Fanuc TP program (LS listing): 190220_hosenrohr_oV2.ls

/PROG  190220_hosenrohr_oV2
/ATTR
COMMENT	= "19-02-22 10:03:29";
PROG_SIZE	= 0;
DEFAULT_GROUP	= 1, 1, *, *, *;
/APPL
    ARC Welding Equipment: 1, *, *, *, *;
/MN
   1:  CALL HOME_ALL;
   1:  UFRAME_NUM = 1;
   1:  UTOOL_NUM = 3;
   1:  COL GUARD ADJUST 150;
   1:  ! -- Layer/Ebene 62 -- !;
   1:  PR[91] = PR[90];
   1:  PR[GP1:91,1] = PR[GP1:90,1] + -0.384;
   1:  PR[GP1:91,2] = PR[GP1:90,2] + 18.027;
   1:  PR[GP1:91,3] = PR[GP1:90,3] + 38.125;
   1:  !Sicherheitspunkt!;
   1:  PR[92] = PR[91];
   1:  PR[92] = PR[GP1:92,3] + 50;
   1:J PR[92];
   1:  !Schweissanfang anfahren!;
   1:L PR[91] R[100]mm/sec CNT100;
   1:  CALL LASER_DRAHT_START;
   1:  PR[GP1:91,1] = PR[GP1:90,1] + -4.016;
   1:  PR[GP1:91,2] = PR[GP1:90,2] + 19.874;
   1:L PR[91] R[100]mm/sec CNT100;
   1:  PR[GP1:91,1] = PR[GP1:90,1] + -8.099;
   1:  PR[GP1:91,2] = PR[GP1:90,2] + 24.627;
   1:L PR[91] R[100]mm/sec CNT100;
   1:  PR[GP1:91,1] = PR[GP1:90,1] + -13.957;
   1:  PR[GP1:91,2] = PR[GP1:90,2] + 29.191;
   1:L PR[91] R[100]mm/sec CNT100;
   1:  PR[GP1:91,1] = PR[GP1:90,1] + -18.277;
   1:  PR[GP1:91,2] = PR[GP1:90,2] + 31.547;
   1:L PR[91] R[100]mm/sec CNT100;
   1:  PR[GP1:91,1] = PR[GP1:90,1] + -22.719;
   1:  PR[GP1:91,2] = PR[GP1:90,2] + 33.113;
   1:L PR[91] R[100]mm/sec CNT100;
   1:  PR[GP1:91,1] = PR[GP1:90,1] + -26.359;
   1:  PR[GP1:91,2] = PR[GP1:90,2] + 34.297;
   1:L PR[91] R[100]mm/sec CNT100;
   1:  PR[GP1:91,1] = PR[GP1:90,1] + -28.832;
   1:  PR[GP1:91,2] = PR[GP1:90,2] + 34.657;
   1:L PR[91] R[100]mm/sec CNT100;
   1:  PR[GP1:91,1] = PR[GP1:90,1] + -36.965;
   1:  PR[GP1:91,2] = PR[GP1:90,2] + 35.069;
   1:L PR[91] R[100]mm/sec CNT100;
   1:  PR[GP1:91,1] = PR[GP1:90,1] + -38.092;
   1:  PR[GP1:91,2] = PR[GP1:90,2] + 35.037;
   1:L PR[91] R[100]mm/sec CNT100;
   1:  PR[GP1:91,1] = PR[GP1:90,1] + -45.127;
   1:  PR[GP1:91,2] = PR[GP1:90,2] + 33.402;
   1:L PR[91] R[100]mm/sec CNT100;
   1:  PR[GP1:91,1] = PR[GP1:90,1] + -48.487;
   1:  PR[GP1:91,2] = PR[GP1:90,2] + 32.649;
   1:L PR[91] R[100]mm/sec CNT100;
   1:  PR[GP1:91,1] = PR[GP1:90,1] + -49.175;
   1:  PR[GP1:91,2] = PR[GP1:90,2] + 32.303;
   1:L PR[91] R[100]mm/sec CNT100;
   1:  PR[GP1:91,1] = PR[GP1:90,1] + -57.619;
   1:  PR[GP1:91,2] = PR[GP1:90,2] + 27.543;
   1:L PR[91] R[100]mm/sec CNT100;
   1:  PR[GP1:91,1] = PR[GP1:90,1] + -59.619;
   1:  PR[GP1:91,2] = PR[GP1:90,2] + 25.581;
   1:L PR[91] R[100]mm/sec CNT100;
   1:  PR[GP1:91,1] = PR[GP1:90,1] + -64.977;
   1:  PR[GP1:91,2] = PR[GP1:90,2] + 19.937;
   1:L PR[91] R[100]mm/sec CNT100;
   1:  PR[GP1:91,1] = PR[GP1:90,1] + -66.878;
   1:  PR[GP1:91,2] = PR[GP1:90,2] + 16.287;
   1:L PR[91] R[100]mm/sec CNT100;
   1:  PR[GP1:91,1] = PR[GP1:90,1] + -69.759;
   1:  PR[GP1:91,2] = PR[GP1:90,2] + 10.455;
   1:L PR[91] R[100]mm/sec CNT100;
   1:  PR[GP1:91,1] = PR[GP1:90,1] + -70.528;
   1:  PR[GP1:91,2] = PR[GP1:90,2] + 5.716;
   1:L PR[91] R[100]mm/sec CNT100;
   1:  PR[GP1:91,1] = PR[GP1:90,1] + -70.620;
   1:  PR[GP1:91,2] = PR[GP1:90,2] + 5.247;
   1:L PR[91] R[100]mm/sec CNT100;
   1:  PR[GP1:91,1] = PR[GP1:90,1] + -71.434;
   1:  PR[GP1:91,2] = PR[GP1:90,2] + -0.068;
   1:L PR[91] R[100]mm/sec CNT100;
   1:  PR[GP1:91,1] = PR[GP1:90,1] + -70.618;
   1:  PR[GP1:91,2] = PR[GP1:90,2] + -4.964;
   1:L PR[91] R[100]mm/sec CNT100;
   1:  PR[GP1:91,1] = PR[GP1:90,1] + -69.758;
   1:  PR[GP1:91,2] = PR[GP1:90,2] + -10.601;
   1:L PR[91] R[100]mm/sec CNT100;
   1:  PR[GP1:91,1] = PR[GP1:90,1] + -66.878;
   1:  PR[GP1:91,2] = PR[GP1:90,2] + -16.431;
   1:L PR[91] R[100]mm/sec CNT100;
   1:  PR[GP1:91,1] = PR[GP1:90,1] + -64.977;
   1:  PR[GP1:91,2] = PR[GP1:90,2] + -20.081;
   1:L PR[91] R[100]mm/sec CNT100;
   1:  PR[GP1:91,1] = PR[GP1:90,1] + -59.619;
   1:  PR[GP1:91,2] = PR[GP1:90,2] + -25.725;
   1:L PR[91] R[100]mm/sec CNT100;
   1:  PR[GP1:91,1] = PR[GP1:90,1] + -57.619;
   1:  PR[GP1:91,2] = PR[GP1:90,2] + -27.687;
   1:L PR[91] R[100]mm/sec CNT100;
   1:  PR[GP1:91,1] = PR[GP1:90,1] + -49.175;
   1:  PR[GP1:91,2] = PR[GP1:90,2] + -32.447;
   1:L PR[91] R[100]mm/sec CNT100;
   1:  PR[GP1:91,1] = PR[GP1:90,1] + -48.487;
   1:  PR[GP1:91,2] = PR[GP1:90,2] + -32.793;
   1:L PR[91] R[100]mm/sec CNT100;
   1:  PR[GP1:91,1] = PR[GP1:90,1] + -45.126;
   1:  PR[GP1:91,2] = PR[GP1:90,2] + -33.546;
   1:L PR[91] R[100]mm/sec CNT100;
   1:  PR[GP1:91,1] = PR[GP1:90,1] + -38.859;
   1:  PR[GP1:91,2] = PR[GP1:90,2] + -35.021;
   1:L PR[91] R[100]mm/sec CNT100;
   1:  PR[GP1:91,1] = PR[GP1:90,1] + -38.098;
   1:  PR[GP1:91,2] = PR[GP1:90,2] + -35.181;
   1:L PR[91] R[100]mm/sec CNT100;
   1:  PR[GP1:91,1] = PR[GP1:90,1] + -36.965;
   1:  PR[GP1:91,2] = PR[GP1:90,2] + -35.213;
   1:L PR[91] R[100]mm/sec CNT100;
   1:  PR[GP1:91,1] = PR[GP1:90,1] + -28.832;
   1:  PR[GP1:91,2] = PR[GP1:90,2] + -34.801;
   1:L PR[91] R[100]mm/sec CNT100;
   1:  PR[GP1:91,1] = PR[GP1:90,1] + -26.368;
   1:  PR[GP1:91,2] = PR[GP1:90,2] + -34.443;
   1:L PR[91] R[100]mm/sec CNT100;
   1:  PR[GP1:91,1] = PR[GP1:90,1] + -21.518;
   1:  PR[GP1:91,2] = PR[GP1:90,2] + -32.707;
   1:L PR[91] R[100]mm/sec CNT100;
   1:  PR[GP1:91,1] = PR[GP1:90,1] + -18.268;
   1:  PR[GP1:91,2] = PR[GP1:90,2] + -31.686;
   1:L PR[91] R[100]mm/sec CNT100;
   1:  PR[GP1:91,1] = PR[GP1:90,1] + -13.949;
   1:  PR[GP1:91,2] = PR[GP1:90,2] + -29.331;
   1:L PR[91] R[100]mm/sec CNT100;
   1:  PR[GP1:91,1] = PR[GP1:90,1] + -12.372;
   1:  PR[GP1:91,2] = PR[GP1:90,2] + -28.176;
   1:L PR[91] R[100]mm/sec CNT100;
   1:  PR[GP1:91,1] = PR[GP1:90,1] + -8.101;
   1:  PR[GP1:91,2] = PR[GP1:90,2] + -24.773;
   1:L PR[91] R[100]mm/sec CNT100;
   1:  PR[GP1:91,1] = PR[GP1:90,1] + -3.961;
   1:  PR[GP1:91,2] = PR[GP1:90,2] + -19.964;
   1:L PR[91] R[100]mm/sec CNT100;
   1:  PR[GP1:91,1] = PR[GP1:90,1] + -3.637;
   1:  PR[GP1:91,2] = PR[GP1:90,2] + -19.895;
   1:L PR[91] R[100]mm/sec CNT100;
   1:  PR[GP1:91,1] = PR[GP1:90,1] + 0.136;
   1:  PR[GP1:91,2] = PR[GP1:90,2] + -17.894;
   1:L PR[91] R[100]mm/sec CNT100;
   1:  PR[GP1:91,1] = PR[GP1:90,1] + 0.611;
   1:  PR[GP1:91,2] = PR[GP1:90,2] + -18.171;
   1:L PR[91] R[100]mm/sec CNT100;
   1:  PR[GP1:91,1] = PR[GP1:90,1] + 4.242;
   1:  PR[GP1:91,2] = PR[GP1:90,2] + -20.026;
   1:L PR[91] R[100]mm/sec CNT100;
   1:  PR[GP1:91,1] = PR[GP1:90,1] + 8.362;
   1:  PR[GP1:91,2] = PR[GP1:90,2] + -24.817;
   1:L PR[91] R[100]mm/sec CNT100;
   1:  PR[GP1:91,1] = PR[GP1:90,1] + 14.189;
   1:  PR[GP1:91,2] = PR[GP1:90,2] + -29.353;
   1:L PR[91] R[100]mm/sec CNT100;
   1:  PR[GP1:91,1] = PR[GP1:90,1] + 18.481;
   1:  PR[GP1:91,2] = PR[GP1:90,2] + -31.687;
   1:L PR[91] R[100]mm/sec CNT100;
   1:  PR[GP1:91,1] = PR[GP1:90,1] + 22.922;
   1:  PR[GP1:91,2] = PR[GP1:90,2] + -33.252;
   1:L PR[91] R[100]mm/sec CNT100;
   1:  PR[GP1:91,1] = PR[GP1:90,1] + 26.570;
   1:  PR[GP1:91,2] = PR[GP1:90,2] + -34.439;
   1:L PR[91] R[100]mm/sec CNT100;
   1:  PR[GP1:91,1] = PR[GP1:90,1] + 29.041;
   1:  PR[GP1:91,2] = PR[GP1:90,2] + -34.800;
   1:L PR[91] R[100]mm/sec CNT100;
   1:  PR[GP1:91,1] = PR[GP1:90,1] + 37.175;
   1:  PR[GP1:91,2] = PR[GP1:90,2] + -35.214;
   1:L PR[91] R[100]mm/sec CNT100;
   1:  PR[GP1:91,1] = PR[GP1:90,1] + 38.299;
   1:  PR[GP1:91,2] = PR[GP1:90,2] + -35.183;
   1:L PR[91] R[100]mm/sec CNT100;
   1:  PR[GP1:91,1] = PR[GP1:90,1] + 45.340;
   1:  PR[GP1:91,2] = PR[GP1:90,2] + -33.544;
   1:L PR[91] R[100]mm/sec CNT100;
   1:  PR[GP1:91,1] = PR[GP1:90,1] + 48.700;
   1:  PR[GP1:91,2] = PR[GP1:90,2] + -32.790;
   1:L PR[91] R[100]mm/sec CNT100;
   1:  PR[GP1:91,1] = PR[GP1:90,1] + 49.388;
   1:  PR[GP1:91,2] = PR[GP1:90,2] + -32.445;
   1:L PR[91] R[100]mm/sec CNT100;
   1:  PR[GP1:91,1] = PR[GP1:90,1] + 57.830;
   1:  PR[GP1:91,2] = PR[GP1:90,2] + -27.694;
   1:L PR[91] R[100]mm/sec CNT100;
   1:  PR[GP1:91,1] = PR[GP1:90,1] + 59.830;
   1:  PR[GP1:91,2] = PR[GP1:90,2] + -25.729;
   1:L PR[91] R[100]mm/sec CNT100;
   1:  PR[GP1:91,1] = PR[GP1:90,1] + 65.189;
   1:  PR[GP1:91,2] = PR[GP1:90,2] + -20.068;
   1:L PR[91] R[100]mm/sec CNT100;
   1:  PR[GP1:91,1] = PR[GP1:90,1] + 67.091;
   1:  PR[GP1:91,2] = PR[GP1:90,2] + -16.427;
   1:L PR[91] R[100]mm/sec CNT100;
   1:  PR[GP1:91,1] = PR[GP1:90,1] + 69.972;
   1:  PR[GP1:91,2] = PR[GP1:90,2] + -10.623;
   1:L PR[91] R[100]mm/sec CNT100;
   1:  PR[GP1:91,1] = PR[GP1:90,1] + 70.741;
   1:  PR[GP1:91,2] = PR[GP1:90,2] + -5.877;
   1:L PR[91] R[100]mm/sec CNT100;
   1:  PR[GP1:91,1] = PR[GP1:90,1] + 70.833;
   1:  PR[GP1:91,2] = PR[GP1:90,2] + -5.406;
   1:L PR[91] R[100]mm/sec CNT100;
   1:  PR[GP1:91,1] = PR[GP1:90,1] + 71.648;
   1:  PR[GP1:91,2] = PR[GP1:90,2] + -0.076;
   1:L PR[91] R[100]mm/sec CNT100;
   1:  PR[GP1:91,1] = PR[GP1:90,1] + 70.831;
   1:  PR[GP1:91,2] = PR[GP1:90,2] + 4.828;
   1:L PR[91] R[100]mm/sec CNT100;
   1:  PR[GP1:91,1] = PR[GP1:90,1] + 69.971;
   1:  PR[GP1:91,2] = PR[GP1:90,2] + 10.481;
   1:L PR[91] R[100]mm/sec CNT100;
   1:  PR[GP1:91,1] = PR[GP1:90,1] + 67.091;
   1:  PR[GP1:91,2] = PR[GP1:90,2] + 16.283;
   1:L PR[91] R[100]mm/sec CNT100;
   1:  PR[GP1:91,1] = PR[GP1:90,1] + 65.189;
   1:  PR[GP1:91,2] = PR[GP1:90,2] + 19.924;
   1:L PR[91] R[100]mm/sec CNT100;
   1:  PR[GP1:91,1] = PR[GP1:90,1] + 59.830;
   1:  PR[GP1:91,2] = PR[GP1:90,2] + 25.585;
   1:L PR[91] R[100]mm/sec CNT100;
   1:  PR[GP1:91,1] = PR[GP1:90,1] + 57.830;
   1:  PR[GP1:91,2] = PR[GP1:90,2] + 27.550;
   1:L PR[91] R[100]mm/sec CNT100;
   1:  PR[GP1:91,1] = PR[GP1:90,1] + 49.388;
   1:  PR[GP1:91,2] = PR[GP1:90,2] + 32.301;
   1:L PR[91] R[100]mm/sec CNT100;
   1:  PR[GP1:91,1] = PR[GP1:90,1] + 48.700;
   1:  PR[GP1:91,2] = PR[GP1:90,2] + 32.646;
   1:L PR[91] R[100]mm/sec CNT100;
   1:  PR[GP1:91,1] = PR[GP1:90,1] + 45.339;
   1:  PR[GP1:91,2] = PR[GP1:90,2] + 33.400;
   1:L PR[91] R[100]mm/sec CNT100;
   1:  PR[GP1:91,1] = PR[GP1:90,1] + 39.068;
   1:  PR[GP1:91,2] = PR[GP1:90,2] + 34.879;
   1:L PR[91] R[100]mm/sec CNT100;
   1:  PR[GP1:91,1] = PR[GP1:90,1] + 38.306;
   1:  PR[GP1:91,2] = PR[GP1:90,2] + 35.039;
   1:L PR[91] R[100]mm/sec CNT100;
   1:  PR[GP1:91,1] = PR[GP1:90,1] + 37.175;
   1:  PR[GP1:91,2] = PR[GP1:90,2] + 35.070;
   1:L PR[91] R[100]mm/sec CNT100;
   1:  PR[GP1:91,1] = PR[GP1:90,1] + 29.041;
   1:  PR[GP1:91,2] = PR[GP1:90,2] + 34.656;
   1:L PR[91] R[100]mm/sec CNT100;
   1:  PR[GP1:91,1] = PR[GP1:90,1] + 26.579;
   1:  PR[GP1:91,2] = PR[GP1:90,2] + 34.296;
   1:L PR[91] R[100]mm/sec CNT100;
   1:  PR[GP1:91,1] = PR[GP1:90,1] + 21.729;
   1:  PR[GP1:91,2] = PR[GP1:90,2] + 32.563;
   1:L PR[91] R[100]mm/sec CNT100;
   1:  PR[GP1:91,1] = PR[GP1:90,1] + 18.472;
   1:  PR[GP1:91,2] = PR[GP1:90,2] + 31.539;
   1:L PR[91] R[100]mm/sec CNT100;
   1:  PR[GP1:91,1] = PR[GP1:90,1] + 14.182;
   1:  PR[GP1:91,2] = PR[GP1:90,2] + 29.205;
   1:L PR[91] R[100]mm/sec CNT100;
   1:  PR[GP1:91,1] = PR[GP1:90,1] + 12.601;
   1:  PR[GP1:91,2] = PR[GP1:90,2] + 28.047;
   1:L PR[91] R[100]mm/sec CNT100;
   1:  PR[GP1:91,1] = PR[GP1:90,1] + 8.365;
   1:  PR[GP1:91,2] = PR[GP1:90,2] + 24.676;
   1:L PR[91] R[100]mm/sec CNT100;
   1:  PR[GP1:91,1] = PR[GP1:90,1] + 4.242;
   1:  PR[GP1:91,2] = PR[GP1:90,2] + 19.873;
   1:L PR[91] R[100]mm/sec CNT100;
   1:  PR[GP1:91,1] = PR[GP1:90,1] + 0.084;
   1:  PR[GP1:91,2] = PR[GP1:90,2] + 17.753;
   1:L PR[91] R[100]mm/sec CNT100;
   1:  ! -- Layer/Ebene 63 -- !;
   1:  PR[91] = PR[90];
   1:  PR[GP1:91,1] = PR[GP1:90,1] + -0.147;
   1:  PR[GP1:91,2] = PR[GP1:90,2] + 18.208;
   1:  PR[GP1:91,3] = PR[GP1:90,3] + 38.735;
   1:L PR[91] R[100]mm/sec CNT100;
   1:  PR[GP1:91,1] = PR[GP1:90,1] + -3.986;
   1:  PR[GP1:91,2] = PR[GP1:90,2] + 20.161;
   1:L PR[91] R[100]mm/sec CNT100;
   1:  PR[GP1:91,1] = PR[GP1:90,1] + -7.934;
   1:  PR[GP1:91,2] = PR[GP1:90,2] + 24.750;
   1:L PR[91] R[100]mm/sec CNT100;
   1:  PR[GP1:91,1] = PR[GP1:90,1] + -13.454;
   1:  PR[GP1:91,2] = PR[GP1:90,2] + 29.065;
   1:L PR[91] R[100]mm/sec CNT100;
   1:  PR[GP1:91,1] = PR[GP1:90,1] + -18.260;
   1:  PR[GP1:91,2] = PR[GP1:90,2] + 31.685;
   1:L PR[91] R[100]mm/sec CNT100;
   1:  PR[GP1:91,1] = PR[GP1:90,1] + -21.778;
   1:  PR[GP1:91,2] = PR[GP1:90,2] + 32.926;
   1:L PR[91] R[100]mm/sec CNT100;
   1:  PR[GP1:91,1] = PR[GP1:90,1] + -26.058;
   1:  PR[GP1:91,2] = PR[GP1:90,2] + 34.319;
   1:L PR[91] R[100]mm/sec CNT100;
   1:  PR[GP1:91,1] = PR[GP1:90,1] + -28.972;
   1:  PR[GP1:91,2] = PR[GP1:90,2] + 34.743;
   1:L PR[91] R[100]mm/sec CNT100;
   1:  PR[GP1:91,1] = PR[GP1:90,1] + -36.314;
   1:  PR[GP1:91,2] = PR[GP1:90,2] + 35.115;
   1:L PR[91] R[100]mm/sec CNT100;
   1:  PR[GP1:91,1] = PR[GP1:90,1] + -37.972;
   1:  PR[GP1:91,2] = PR[GP1:90,2] + 35.068;
   1:L PR[91] R[100]mm/sec CNT100;
   1:  PR[GP1:91,1] = PR[GP1:90,1] + -48.463;
   1:  PR[GP1:91,2] = PR[GP1:90,2] + 32.632;
   1:L PR[91] R[100]mm/sec CNT100;
   1:  PR[GP1:91,1] = PR[GP1:90,1] + -57.569;
   1:  PR[GP1:91,2] = PR[GP1:90,2] + 27.505;
   1:L PR[91] R[100]mm/sec CNT100;
   1:  PR[GP1:91,1] = PR[GP1:90,1] + -59.075;
   1:  PR[GP1:91,2] = PR[GP1:90,2] + 26.027;
   1:L PR[91] R[100]mm/sec CNT100;
   1:  PR[GP1:91,1] = PR[GP1:90,1] + -64.892;
   1:  PR[GP1:91,2] = PR[GP1:90,2] + 19.900;
   1:L PR[91] R[100]mm/sec CNT100;
   1:  PR[GP1:91,1] = PR[GP1:90,1] + -66.497;
   1:  PR[GP1:91,2] = PR[GP1:90,2] + 16.818;
   1:L PR[91] R[100]mm/sec CNT100;
   1:  PR[GP1:91,1] = PR[GP1:90,1] + -69.651;
   1:  PR[GP1:91,2] = PR[GP1:90,2] + 10.434;
   1:L PR[91] R[100]mm/sec CNT100;
   1:  PR[GP1:91,1] = PR[GP1:90,1] + -70.323;
   1:  PR[GP1:91,2] = PR[GP1:90,2] + 6.290;
   1:L PR[91] R[100]mm/sec CNT100;
   1:  PR[GP1:91,1] = PR[GP1:90,1] + -70.403;
   1:  PR[GP1:91,2] = PR[GP1:90,2] + 5.879;
   1:L PR[91] R[100]mm/sec CNT100;
   1:  PR[GP1:91,1] = PR[GP1:90,1] + -71.315;
   1:  PR[GP1:91,2] = PR[GP1:90,2] + -0.068;
   1:L PR[91] R[100]mm/sec CNT100;
   1:  PR[GP1:91,1] = PR[GP1:90,1] + -70.592;
   1:  PR[GP1:91,2] = PR[GP1:90,2] + -4.409;
   1:L PR[91] R[100]mm/sec CNT100;
   1:  PR[GP1:91,1] = PR[GP1:90,1] + -69.650;
   1:  PR[GP1:91,2] = PR[GP1:90,2] + -10.580;
   1:L PR[91] R[100]mm/sec CNT100;
   1:  PR[GP1:91,1] = PR[GP1:90,1] + -66.497;
   1:  PR[GP1:91,2] = PR[GP1:90,2] + -16.962;
   1:L PR[91] R[100]mm/sec CNT100;
   1:  PR[GP1:91,1] = PR[GP1:90,1] + -64.892;
   1:  PR[GP1:91,2] = PR[GP1:90,2] + -20.044;
   1:L PR[91] R[100]mm/sec CNT100;
   1:  PR[GP1:91,1] = PR[GP1:90,1] + -59.075;
   1:  PR[GP1:91,2] = PR[GP1:90,2] + -26.171;
   1:L PR[91] R[100]mm/sec CNT100;
   1:  PR[GP1:91,1] = PR[GP1:90,1] + -57.569;
   1:  PR[GP1:91,2] = PR[GP1:90,2] + -27.649;
   1:L PR[91] R[100]mm/sec CNT100;
   1:  PR[GP1:91,1] = PR[GP1:90,1] + -48.463;
   1:  PR[GP1:91,2] = PR[GP1:90,2] + -32.777;
   1:L PR[91] R[100]mm/sec CNT100;
   1:  PR[GP1:91,1] = PR[GP1:90,1] + -39.099;
   1:  PR[GP1:91,2] = PR[GP1:90,2] + -34.975;
   1:L PR[91] R[100]mm/sec CNT100;
   1:  PR[GP1:91,1] = PR[GP1:90,1] + -37.979;
   1:  PR[GP1:91,2] = PR[GP1:90,2] + -35.211;
   1:L PR[91] R[100]mm/sec CNT100;
   1:  PR[GP1:91,1] = PR[GP1:90,1] + -36.314;
   1:  PR[GP1:91,2] = PR[GP1:90,2] + -35.259;
   1:L PR[91] R[100]mm/sec CNT100;
   1:  PR[GP1:91,1] = PR[GP1:90,1] + -28.972;
   1:  PR[GP1:91,2] = PR[GP1:90,2] + -34.887;
   1:L PR[91] R[100]mm/sec CNT100;
   1:  PR[GP1:91,1] = PR[GP1:90,1] + -26.066;
   1:  PR[GP1:91,2] = PR[GP1:90,2] + -34.464;
   1:L PR[91] R[100]mm/sec CNT100;
   1:  PR[GP1:91,1] = PR[GP1:90,1] + -21.865;
   1:  PR[GP1:91,2] = PR[GP1:90,2] + -32.960;
   1:L PR[91] R[100]mm/sec CNT100;
   1:  PR[GP1:91,1] = PR[GP1:90,1] + -18.251;
   1:  PR[GP1:91,2] = PR[GP1:90,2] + -31.824;
   1:L PR[91] R[100]mm/sec CNT100;
   1:  PR[GP1:91,1] = PR[GP1:90,1] + -13.445;
   1:  PR[GP1:91,2] = PR[GP1:90,2] + -29.204;
   1:L PR[91] R[100]mm/sec CNT100;
   1:  PR[GP1:91,1] = PR[GP1:90,1] + -12.545;
   1:  PR[GP1:91,2] = PR[GP1:90,2] + -28.544;
   1:L PR[91] R[100]mm/sec CNT100;
   1:  PR[GP1:91,1] = PR[GP1:90,1] + -9.672;
   1:  PR[GP1:91,2] = PR[GP1:90,2] + -26.256;
   1:L PR[91] R[100]mm/sec CNT100;
   1:  PR[GP1:91,1] = PR[GP1:90,1] + -7.920;
   1:  PR[GP1:91,2] = PR[GP1:90,2] + -24.884;
   1:L PR[91] R[100]mm/sec CNT100;
   1:  PR[GP1:91,1] = PR[GP1:90,1] + -3.931;
   1:  PR[GP1:91,2] = PR[GP1:90,2] + -20.257;
   1:L PR[91] R[100]mm/sec CNT100;
   1:  PR[GP1:91,1] = PR[GP1:90,1] + -3.470;
   1:  PR[GP1:91,2] = PR[GP1:90,2] + -20.158;
   1:L PR[91] R[100]mm/sec CNT100;
   1:  PR[GP1:91,1] = PR[GP1:90,1] + 0.146;
   1:  PR[GP1:91,2] = PR[GP1:90,2] + -18.242;
   1:L PR[91] R[100]mm/sec CNT100;
   1:  PR[GP1:91,1] = PR[GP1:90,1] + 4.212;
   1:  PR[GP1:91,2] = PR[GP1:90,2] + -20.319;
   1:L PR[91] R[100]mm/sec CNT100;
   1:  PR[GP1:91,1] = PR[GP1:90,1] + 8.183;
   1:  PR[GP1:91,2] = PR[GP1:90,2] + -24.930;
   1:L PR[91] R[100]mm/sec CNT100;
   1:  PR[GP1:91,1] = PR[GP1:90,1] + 13.688;
   1:  PR[GP1:91,2] = PR[GP1:90,2] + -29.229;
   1:L PR[91] R[100]mm/sec CNT100;
   1:  PR[GP1:91,1] = PR[GP1:90,1] + 18.463;
   1:  PR[GP1:91,2] = PR[GP1:90,2] + -31.826;
   1:L PR[91] R[100]mm/sec CNT100;
   1:  PR[GP1:91,1] = PR[GP1:90,1] + 21.979;
   1:  PR[GP1:91,2] = PR[GP1:90,2] + -33.064;
   1:L PR[91] R[100]mm/sec CNT100;
   1:  PR[GP1:91,1] = PR[GP1:90,1] + 26.268;
   1:  PR[GP1:91,2] = PR[GP1:90,2] + -34.460;
   1:L PR[91] R[100]mm/sec CNT100;
   1:  PR[GP1:91,1] = PR[GP1:90,1] + 29.180;
   1:  PR[GP1:91,2] = PR[GP1:90,2] + -34.886;
   1:L PR[91] R[100]mm/sec CNT100;
   1:  PR[GP1:91,1] = PR[GP1:90,1] + 36.523;
   1:  PR[GP1:91,2] = PR[GP1:90,2] + -35.259;
   1:L PR[91] R[100]mm/sec CNT100;
   1:  PR[GP1:91,1] = PR[GP1:90,1] + 38.177;
   1:  PR[GP1:91,2] = PR[GP1:90,2] + -35.213;
   1:L PR[91] R[100]mm/sec CNT100;
   1:  PR[GP1:91,1] = PR[GP1:90,1] + 48.676;
   1:  PR[GP1:91,2] = PR[GP1:90,2] + -32.773;
   1:L PR[91] R[100]mm/sec CNT100;
   1:  PR[GP1:91,1] = PR[GP1:90,1] + 57.781;
   1:  PR[GP1:91,2] = PR[GP1:90,2] + -27.655;
   1:L PR[91] R[100]mm/sec CNT100;
   1:  PR[GP1:91,1] = PR[GP1:90,1] + 59.287;
   1:  PR[GP1:91,2] = PR[GP1:90,2] + -26.175;
   1:L PR[91] R[100]mm/sec CNT100;
   1:  PR[GP1:91,1] = PR[GP1:90,1] + 65.104;
   1:  PR[GP1:91,2] = PR[GP1:90,2] + -20.031;
   1:L PR[91] R[100]mm/sec CNT100;
   1:  PR[GP1:91,1] = PR[GP1:90,1] + 66.710;
   1:  PR[GP1:91,2] = PR[GP1:90,2] + -16.955;
   1:L PR[91] R[100]mm/sec CNT100;
   1:  PR[GP1:91,1] = PR[GP1:90,1] + 69.864;
   1:  PR[GP1:91,2] = PR[GP1:90,2] + -10.602;
   1:L PR[91] R[100]mm/sec CNT100;
   1:  PR[GP1:91,1] = PR[GP1:90,1] + 70.536;
   1:  PR[GP1:91,2] = PR[GP1:90,2] + -6.453;
   1:L PR[91] R[100]mm/sec CNT100;
   1:  PR[GP1:91,1] = PR[GP1:90,1] + 70.616;
   1:  PR[GP1:91,2] = PR[GP1:90,2] + -6.041;
   1:L PR[91] R[100]mm/sec CNT100;
   1:  PR[GP1:91,1] = PR[GP1:90,1] + 71.528;
   1:  PR[GP1:91,2] = PR[GP1:90,2] + -0.076;
   1:L PR[91] R[100]mm/sec CNT100;
   1:  PR[GP1:91,1] = PR[GP1:90,1] + 70.804;
   1:  PR[GP1:91,2] = PR[GP1:90,2] + 4.273;
   1:L PR[91] R[100]mm/sec CNT100;
   1:  PR[GP1:91,1] = PR[GP1:90,1] + 69.862;
   1:  PR[GP1:91,2] = PR[GP1:90,2] + 10.461;
   1:L PR[91] R[100]mm/sec CNT100;
   1:  PR[GP1:91,1] = PR[GP1:90,1] + 66.710;
   1:  PR[GP1:91,2] = PR[GP1:90,2] + 16.811;
   1:L PR[91] R[100]mm/sec CNT100;
   1:  PR[GP1:91,1] = PR[GP1:90,1] + 65.104;
   1:  PR[GP1:91,2] = PR[GP1:90,2] + 19.887;
   1:L PR[91] R[100]mm/sec CNT100;
   1:  PR[GP1:91,1] = PR[GP1:90,1] + 59.287;
   1:  PR[GP1:91,2] = PR[GP1:90,2] + 26.031;
   1:L PR[91] R[100]mm/sec CNT100;
   1:  PR[GP1:91,1] = PR[GP1:90,1] + 57.781;
   1:  PR[GP1:91,2] = PR[GP1:90,2] + 27.511;
   1:L PR[91] R[100]mm/sec CNT100;
   1:  PR[GP1:91,1] = PR[GP1:90,1] + 48.676;
   1:  PR[GP1:91,2] = PR[GP1:90,2] + 32.629;
   1:L PR[91] R[100]mm/sec CNT100;
   1:  PR[GP1:91,1] = PR[GP1:90,1] + 39.306;
   1:  PR[GP1:91,2] = PR[GP1:90,2] + 34.833;
   1:L PR[91] R[100]mm/sec CNT100;
   1:  PR[GP1:91,1] = PR[GP1:90,1] + 38.184;
   1:  PR[GP1:91,2] = PR[GP1:90,2] + 35.069;
   1:L PR[91] R[100]mm/sec CNT100;
   1:  PR[GP1:91,1] = PR[GP1:90,1] + 36.523;
   1:  PR[GP1:91,2] = PR[GP1:90,2] + 35.115;
   1:L PR[91] R[100]mm/sec CNT100;
   1:  PR[GP1:91,1] = PR[GP1:90,1] + 29.181;
   1:  PR[GP1:91,2] = PR[GP1:90,2] + 34.742;
   1:L PR[91] R[100]mm/sec CNT100;
   1:  PR[GP1:91,1] = PR[GP1:90,1] + 26.277;
   1:  PR[GP1:91,2] = PR[GP1:90,2] + 34.317;
   1:L PR[91] R[100]mm/sec CNT100;
   1:  PR[GP1:91,1] = PR[GP1:90,1] + 22.076;
   1:  PR[GP1:91,2] = PR[GP1:90,2] + 32.816;
   1:L PR[91] R[100]mm/sec CNT100;
   1:  PR[GP1:91,1] = PR[GP1:90,1] + 18.454;
   1:  PR[GP1:91,2] = PR[GP1:90,2] + 31.677;
   1:L PR[91] R[100]mm/sec CNT100;
   1:  PR[GP1:91,1] = PR[GP1:90,1] + 13.680;
   1:  PR[GP1:91,2] = PR[GP1:90,2] + 29.080;
   1:L PR[91] R[100]mm/sec CNT100;
   1:  PR[GP1:91,1] = PR[GP1:90,1] + 12.775;
   1:  PR[GP1:91,2] = PR[GP1:90,2] + 28.417;
   1:L PR[91] R[100]mm/sec CNT100;
   1:  PR[GP1:91,1] = PR[GP1:90,1] + 9.885;
   1:  PR[GP1:91,2] = PR[GP1:90,2] + 26.118;
   1:L PR[91] R[100]mm/sec CNT100;
   1:  PR[GP1:91,1] = PR[GP1:90,1] + 8.196;
   1:  PR[GP1:91,2] = PR[GP1:90,2] + 24.796;
   1:L PR[91] R[100]mm/sec CNT100;
   1:  PR[GP1:91,1] = PR[GP1:90,1] + 4.193;
   1:  PR[GP1:91,2] = PR[GP1:90,2] + 20.137;
   1:L PR[91] R[100]mm/sec CNT100;
   1:  PR[GP1:91,1] = PR[GP1:90,1] + 3.934;
   1:  PR[GP1:91,2] = PR[GP1:90,2] + 20.034;
   1:L PR[91] R[100]mm/sec CNT100;
   1:  PR[GP1:91,1] = PR[GP1:90,1] + 0.258;
   1:  PR[GP1:91,2] = PR[GP1:90,2] + 18.156;
   1:L PR[91] R[100]mm/sec CNT100;
   1:  ! -- Layer/Ebene 64 -- !;
   1:  PR[91] = PR[90];
   1:  PR[GP1:91,1] = PR[GP1:90,1] + -0.236;
   1:  PR[GP1:91,2] = PR[GP1:90,2] + 18.554;
   1:  PR[GP1:91,3] = PR[GP1:90,3] + 39.345;
   1:L PR[91] R[100]mm/sec CNT100;
   1:  PR[GP1:91,1] = PR[GP1:90,1] + -3.957;
   1:  PR[GP1:91,2] = PR[GP1:90,2] + 20.447;
   1:L PR[91] R[100]mm/sec CNT100;
   1:  PR[GP1:91,1] = PR[GP1:90,1] + -7.778;
   1:  PR[GP1:91,2] = PR[GP1:90,2] + 24.890;
   1:L PR[91] R[100]mm/sec CNT100;
   1:  PR[GP1:91,1] = PR[GP1:90,1] + -12.950;
   1:  PR[GP1:91,2] = PR[GP1:90,2] + 28.938;
   1:L PR[91] R[100]mm/sec CNT100;
   1:  PR[GP1:91,1] = PR[GP1:90,1] + -18.243;
   1:  PR[GP1:91,2] = PR[GP1:90,2] + 31.824;
   1:L PR[91] R[100]mm/sec CNT100;
   1:  PR[GP1:91,1] = PR[GP1:90,1] + -20.838;
   1:  PR[GP1:91,2] = PR[GP1:90,2] + 32.739;
   1:L PR[91] R[100]mm/sec CNT100;
   1:  PR[GP1:91,1] = PR[GP1:90,1] + -25.756;
   1:  PR[GP1:91,2] = PR[GP1:90,2] + 34.340;
   1:L PR[91] R[100]mm/sec CNT100;
   1:  PR[GP1:91,1] = PR[GP1:90,1] + -29.112;
   1:  PR[GP1:91,2] = PR[GP1:90,2] + 34.828;
   1:L PR[91] R[100]mm/sec CNT100;
   1:  PR[GP1:91,1] = PR[GP1:90,1] + -35.663;
   1:  PR[GP1:91,2] = PR[GP1:90,2] + 35.160;
   1:L PR[91] R[100]mm/sec CNT100;
   1:  PR[GP1:91,1] = PR[GP1:90,1] + -37.853;
   1:  PR[GP1:91,2] = PR[GP1:90,2] + 35.098;
   1:L PR[91] R[100]mm/sec CNT100;
   1:  PR[GP1:91,1] = PR[GP1:90,1] + -48.166;
   1:  PR[GP1:91,2] = PR[GP1:90,2] + 32.708;
   1:L PR[91] R[100]mm/sec CNT100;
   1:  PR[GP1:91,1] = PR[GP1:90,1] + -48.426;
   1:  PR[GP1:91,2] = PR[GP1:90,2] + 32.606;
   1:L PR[91] R[100]mm/sec CNT100;
   1:  PR[GP1:91,1] = PR[GP1:90,1] + -57.519;
   1:  PR[GP1:91,2] = PR[GP1:90,2] + 27.467;
   1:L PR[91] R[100]mm/sec CNT100;
   1:  PR[GP1:91,1] = PR[GP1:90,1] + -58.532;
   1:  PR[GP1:91,2] = PR[GP1:90,2] + 26.472;
   1:L PR[91] R[100]mm/sec CNT100;
   1:  PR[GP1:91,1] = PR[GP1:90,1] + -64.807;
   1:  PR[GP1:91,2] = PR[GP1:90,2] + 19.863;
   1:L PR[91] R[100]mm/sec CNT100;
   1:  PR[GP1:91,1] = PR[GP1:90,1] + -66.116;
   1:  PR[GP1:91,2] = PR[GP1:90,2] + 17.349;
   1:L PR[91] R[100]mm/sec CNT100;
   1:  PR[GP1:91,1] = PR[GP1:90,1] + -69.543;
   1:  PR[GP1:91,2] = PR[GP1:90,2] + 10.413;
   1:L PR[91] R[100]mm/sec CNT100;
   1:  PR[GP1:91,1] = PR[GP1:90,1] + -70.118;
   1:  PR[GP1:91,2] = PR[GP1:90,2] + 6.865;
   1:L PR[91] R[100]mm/sec CNT100;
   1:  PR[GP1:91,1] = PR[GP1:90,1] + -70.187;
   1:  PR[GP1:91,2] = PR[GP1:90,2] + 6.512;
   1:L PR[91] R[100]mm/sec CNT100;
   1:  PR[GP1:91,1] = PR[GP1:90,1] + -71.196;
   1:  PR[GP1:91,2] = PR[GP1:90,2] + -0.068;
   1:L PR[91] R[100]mm/sec CNT100;
   1:  PR[GP1:91,1] = PR[GP1:90,1] + -70.565;
   1:  PR[GP1:91,2] = PR[GP1:90,2] + -3.855;
   1:L PR[91] R[100]mm/sec CNT100;
   1:  PR[GP1:91,1] = PR[GP1:90,1] + -69.541;
   1:  PR[GP1:91,2] = PR[GP1:90,2] + -10.560;
   1:L PR[91] R[100]mm/sec CNT100;
   1:  PR[GP1:91,1] = PR[GP1:90,1] + -66.116;
   1:  PR[GP1:91,2] = PR[GP1:90,2] + -17.492;
   1:L PR[91] R[100]mm/sec CNT100;
   1:  PR[GP1:91,1] = PR[GP1:90,1] + -64.807;
   1:  PR[GP1:91,2] = PR[GP1:90,2] + -20.007;
   1:L PR[91] R[100]mm/sec CNT100;
   1:  PR[GP1:91,1] = PR[GP1:90,1] + -58.532;
   1:  PR[GP1:91,2] = PR[GP1:90,2] + -26.616;
   1:L PR[91] R[100]mm/sec CNT100;
   1:  PR[GP1:91,1] = PR[GP1:90,1] + -57.519;
   1:  PR[GP1:91,2] = PR[GP1:90,2] + -27.611;
   1:L PR[91] R[100]mm/sec CNT100;
   1:  PR[GP1:91,1] = PR[GP1:90,1] + -48.610;
   1:  PR[GP1:91,2] = PR[GP1:90,2] + -32.630;
   1:L PR[91] R[100]mm/sec CNT100;
   1:  PR[GP1:91,1] = PR[GP1:90,1] + -48.412;
   1:  PR[GP1:91,2] = PR[GP1:90,2] + -32.755;
   1:L PR[91] R[100]mm/sec CNT100;
   1:  PR[GP1:91,1] = PR[GP1:90,1] + -48.164;
   1:  PR[GP1:91,2] = PR[GP1:90,2] + -32.853;
   1:L PR[91] R[100]mm/sec CNT100;
   1:  PR[GP1:91,1] = PR[GP1:90,1] + -39.339;
   1:  PR[GP1:91,2] = PR[GP1:90,2] + -34.930;
   1:L PR[91] R[100]mm/sec CNT100;
   1:  PR[GP1:91,1] = PR[GP1:90,1] + -37.859;
   1:  PR[GP1:91,2] = PR[GP1:90,2] + -35.242;
   1:L PR[91] R[100]mm/sec CNT100;
   1:  PR[GP1:91,1] = PR[GP1:90,1] + -35.663;
   1:  PR[GP1:91,2] = PR[GP1:90,2] + -35.304;
   1:L PR[91] R[100]mm/sec CNT100;
   1:  PR[GP1:91,1] = PR[GP1:90,1] + -29.112;
   1:  PR[GP1:91,2] = PR[GP1:90,2] + -34.972;
   1:L PR[91] R[100]mm/sec CNT100;
   1:  PR[GP1:91,1] = PR[GP1:90,1] + -25.765;
   1:  PR[GP1:91,2] = PR[GP1:90,2] + -34.485;
   1:L PR[91] R[100]mm/sec CNT100;
   1:  PR[GP1:91,1] = PR[GP1:90,1] + -22.212;
   1:  PR[GP1:91,2] = PR[GP1:90,2] + -33.214;
   1:L PR[91] R[100]mm/sec CNT100;
   1:  PR[GP1:91,1] = PR[GP1:90,1] + -18.234;
   1:  PR[GP1:91,2] = PR[GP1:90,2] + -31.963;
   1:L PR[91] R[100]mm/sec CNT100;
   1:  PR[GP1:91,1] = PR[GP1:90,1] + -12.941;
   1:  PR[GP1:91,2] = PR[GP1:90,2] + -29.077;
   1:L PR[91] R[100]mm/sec CNT100;
   1:  PR[GP1:91,1] = PR[GP1:90,1] + -12.715;
   1:  PR[GP1:91,2] = PR[GP1:90,2] + -28.912;
   1:L PR[91] R[100]mm/sec CNT100;
   1:  PR[GP1:91,1] = PR[GP1:90,1] + -7.747;
   1:  PR[GP1:91,2] = PR[GP1:90,2] + -25.010;
   1:L PR[91] R[100]mm/sec CNT100;
   1:  PR[GP1:91,1] = PR[GP1:90,1] + -3.902;
   1:  PR[GP1:91,2] = PR[GP1:90,2] + -20.550;
   1:L PR[91] R[100]mm/sec CNT100;
   1:  PR[GP1:91,1] = PR[GP1:90,1] + -3.303;
   1:  PR[GP1:91,2] = PR[GP1:90,2] + -20.422;
   1:L PR[91] R[100]mm/sec CNT100;
   1:  PR[GP1:91,1] = PR[GP1:90,1] + 0.187;
   1:  PR[GP1:91,2] = PR[GP1:90,2] + -18.572;
   1:L PR[91] R[100]mm/sec CNT100;
   1:  PR[GP1:91,1] = PR[GP1:90,1] + 4.182;
   1:  PR[GP1:91,2] = PR[GP1:90,2] + -20.612;
   1:L PR[91] R[100]mm/sec CNT100;
   1:  PR[GP1:91,1] = PR[GP1:90,1] + 8.008;
   1:  PR[GP1:91,2] = PR[GP1:90,2] + -25.054;
   1:L PR[91] R[100]mm/sec CNT100;
   1:  PR[GP1:91,1] = PR[GP1:90,1] + 13.186;
   1:  PR[GP1:91,2] = PR[GP1:90,2] + -29.104;
   1:L PR[91] R[100]mm/sec CNT100;
   1:  PR[GP1:91,1] = PR[GP1:90,1] + 18.445;
   1:  PR[GP1:91,2] = PR[GP1:90,2] + -31.964;
   1:L PR[91] R[100]mm/sec CNT100;
   1:  PR[GP1:91,1] = PR[GP1:90,1] + 21.037;
   1:  PR[GP1:91,2] = PR[GP1:90,2] + -32.877;
   1:L PR[91] R[100]mm/sec CNT100;
   1:  PR[GP1:91,1] = PR[GP1:90,1] + 25.967;
   1:  PR[GP1:91,2] = PR[GP1:90,2] + -34.481;
   1:L PR[91] R[100]mm/sec CNT100;
   1:  PR[GP1:91,1] = PR[GP1:90,1] + 29.320;
   1:  PR[GP1:91,2] = PR[GP1:90,2] + -34.971;
   1:L PR[91] R[100]mm/sec CNT100;
   1:  PR[GP1:91,1] = PR[GP1:90,1] + 35.871;
   1:  PR[GP1:91,2] = PR[GP1:90,2] + -35.305;
   1:L PR[91] R[100]mm/sec CNT100;
   1:  PR[GP1:91,1] = PR[GP1:90,1] + 38.055;
   1:  PR[GP1:91,2] = PR[GP1:90,2] + -35.244;
   1:L PR[91] R[100]mm/sec CNT100;
   1:  PR[GP1:91,1] = PR[GP1:90,1] + 48.376;
   1:  PR[GP1:91,2] = PR[GP1:90,2] + -32.850;
   1:L PR[91] R[100]mm/sec CNT100;
   1:  PR[GP1:91,1] = PR[GP1:90,1] + 48.639;
   1:  PR[GP1:91,2] = PR[GP1:90,2] + -32.747;
   1:L PR[91] R[100]mm/sec CNT100;
   1:  PR[GP1:91,1] = PR[GP1:90,1] + 57.731;
   1:  PR[GP1:91,2] = PR[GP1:90,2] + -27.617;
   1:L PR[91] R[100]mm/sec CNT100;
   1:  PR[GP1:91,1] = PR[GP1:90,1] + 58.744;
   1:  PR[GP1:91,2] = PR[GP1:90,2] + -26.621;
   1:L PR[91] R[100]mm/sec CNT100;
   1:  PR[GP1:91,1] = PR[GP1:90,1] + 65.019;
   1:  PR[GP1:91,2] = PR[GP1:90,2] + -19.993;
   1:L PR[91] R[100]mm/sec CNT100;
   1:  PR[GP1:91,1] = PR[GP1:90,1] + 66.329;
   1:  PR[GP1:91,2] = PR[GP1:90,2] + -17.484;
   1:L PR[91] R[100]mm/sec CNT100;
   1:  PR[GP1:91,1] = PR[GP1:90,1] + 69.756;
   1:  PR[GP1:91,2] = PR[GP1:90,2] + -10.582;
   1:L PR[91] R[100]mm/sec CNT100;
   1:  PR[GP1:91,1] = PR[GP1:90,1] + 70.331;
   1:  PR[GP1:91,2] = PR[GP1:90,2] + -7.029;
   1:L PR[91] R[100]mm/sec CNT100;
   1:  PR[GP1:91,1] = PR[GP1:90,1] + 70.400;
   1:  PR[GP1:91,2] = PR[GP1:90,2] + -6.675;
   1:L PR[91] R[100]mm/sec CNT100;
   1:  PR[GP1:91,1] = PR[GP1:90,1] + 71.409;
   1:  PR[GP1:91,2] = PR[GP1:90,2] + -0.076;
   1:L PR[91] R[100]mm/sec CNT100;
   1:  PR[GP1:91,1] = PR[GP1:90,1] + 70.778;
   1:  PR[GP1:91,2] = PR[GP1:90,2] + 3.717;
   1:L PR[91] R[100]mm/sec CNT100;
   1:  PR[GP1:91,1] = PR[GP1:90,1] + 69.754;
   1:  PR[GP1:91,2] = PR[GP1:90,2] + 10.441;
   1:L PR[91] R[100]mm/sec CNT100;
   1:  PR[GP1:91,1] = PR[GP1:90,1] + 66.329;
   1:  PR[GP1:91,2] = PR[GP1:90,2] + 17.340;
   1:L PR[91] R[100]mm/sec CNT100;
   1:  PR[GP1:91,1] = PR[GP1:90,1] + 65.019;
   1:  PR[GP1:91,2] = PR[GP1:90,2] + 19.849;
   1:L PR[91] R[100]mm/sec CNT100;
   1:  PR[GP1:91,1] = PR[GP1:90,1] + 58.744;
   1:  PR[GP1:91,2] = PR[GP1:90,2] + 26.477;
   1:L PR[91] R[100]mm/sec CNT100;
   1:  PR[GP1:91,1] = PR[GP1:90,1] + 57.731;
   1:  PR[GP1:91,2] = PR[GP1:90,2] + 27.473;
   1:L PR[91] R[100]mm/sec CNT100;
   1:  PR[GP1:91,1] = PR[GP1:90,1] + 48.821;
   1:  PR[GP1:91,2] = PR[GP1:90,2] + 32.485;
   1:L PR[91] R[100]mm/sec CNT100;
   1:  PR[GP1:91,1] = PR[GP1:90,1] + 48.625;
   1:  PR[GP1:91,2] = PR[GP1:90,2] + 32.608;
   1:L PR[91] R[100]mm/sec CNT100;
   1:  PR[GP1:91,1] = PR[GP1:90,1] + 48.375;
   1:  PR[GP1:91,2] = PR[GP1:90,2] + 32.706;
   1:L PR[91] R[100]mm/sec CNT100;
   1:  PR[GP1:91,1] = PR[GP1:90,1] + 39.544;
   1:  PR[GP1:91,2] = PR[GP1:90,2] + 34.788;
   1:L PR[91] R[100]mm/sec CNT100;
   1:  PR[GP1:91,1] = PR[GP1:90,1] + 38.061;
   1:  PR[GP1:91,2] = PR[GP1:90,2] + 35.100;
   1:L PR[91] R[100]mm/sec CNT100;
   1:  PR[GP1:91,1] = PR[GP1:90,1] + 35.871;
   1:  PR[GP1:91,2] = PR[GP1:90,2] + 35.161;
   1:L PR[91] R[100]mm/sec CNT100;
   1:  PR[GP1:91,1] = PR[GP1:90,1] + 29.320;
   1:  PR[GP1:91,2] = PR[GP1:90,2] + 34.827;
   1:L PR[91] R[100]mm/sec CNT100;
   1:  PR[GP1:91,1] = PR[GP1:90,1] + 25.975;
   1:  PR[GP1:91,2] = PR[GP1:90,2] + 34.338;
   1:L PR[91] R[100]mm/sec CNT100;
   1:  PR[GP1:91,1] = PR[GP1:90,1] + 22.423;
   1:  PR[GP1:91,2] = PR[GP1:90,2] + 33.068;
   1:L PR[91] R[100]mm/sec CNT100;
   1:  PR[GP1:91,1] = PR[GP1:90,1] + 18.436;
   1:  PR[GP1:91,2] = PR[GP1:90,2] + 31.815;
   1:L PR[91] R[100]mm/sec CNT100;
   1:  PR[GP1:91,1] = PR[GP1:90,1] + 13.178;
   1:  PR[GP1:91,2] = PR[GP1:90,2] + 28.955;
   1:L PR[91] R[100]mm/sec CNT100;
   1:  PR[GP1:91,1] = PR[GP1:90,1] + 12.946;
   1:  PR[GP1:91,2] = PR[GP1:90,2] + 28.785;
   1:L PR[91] R[100]mm/sec CNT100;
   1:  PR[GP1:91,1] = PR[GP1:90,1] + 8.039;
   1:  PR[GP1:91,2] = PR[GP1:90,2] + 24.934;
   1:L PR[91] R[100]mm/sec CNT100;
   1:  PR[GP1:91,1] = PR[GP1:90,1] + 4.163;
   1:  PR[GP1:91,2] = PR[GP1:90,2] + 20.423;
   1:L PR[91] R[100]mm/sec CNT100;
   1:  PR[GP1:91,1] = PR[GP1:90,1] + 3.845;
   1:  PR[GP1:91,2] = PR[GP1:90,2] + 20.298;
   1:L PR[91] R[100]mm/sec CNT100;
   1:  PR[GP1:91,1] = PR[GP1:90,1] + 0.300;
   1:  PR[GP1:91,2] = PR[GP1:90,2] + 18.486;
   1:L PR[91] R[100]mm/sec CNT100;
   1:  ! -- Layer/Ebene 65 -- !;
   1:  PR[91] = PR[90];
   1:  PR[GP1:91,1] = PR[GP1:90,1] + -0.325;
   1:  PR[GP1:91,2] = PR[GP1:90,2] + 18.901;
   1:  PR[GP1:91,3] = PR[GP1:90,3] + 39.955;
   1:L PR[91] R[100]mm/sec CNT100;
   1:  PR[GP1:91,1] = PR[GP1:90,1] + -3.928;
   1:  PR[GP1:91,2] = PR[GP1:90,2] + 20.734;
   1:L PR[91] R[100]mm/sec CNT100;
   1:  PR[GP1:91,1] = PR[GP1:90,1] + -7.622;
   1:  PR[GP1:91,2] = PR[GP1:90,2] + 25.029;
   1:L PR[91] R[100]mm/sec CNT100;
   1:  PR[GP1:91,1] = PR[GP1:90,1] + -12.579;
   1:  PR[GP1:91,2] = PR[GP1:90,2] + 28.912;
   1:L PR[91] R[100]mm/sec CNT100;
   1:  PR[GP1:91,1] = PR[GP1:90,1] + -12.606;
   1:  PR[GP1:91,2] = PR[GP1:90,2] + 28.931;
   1:L PR[91] R[100]mm/sec CNT100;
   1:  PR[GP1:91,1] = PR[GP1:90,1] + -14.058;
   1:  PR[GP1:91,2] = PR[GP1:90,2] + 29.690;
   1:L PR[91] R[100]mm/sec CNT100;
   1:  PR[GP1:91,1] = PR[GP1:90,1] + -18.226;
   1:  PR[GP1:91,2] = PR[GP1:90,2] + 31.963;
   1:L PR[91] R[100]mm/sec CNT100;
   1:  PR[GP1:91,1] = PR[GP1:90,1] + -19.897;
   1:  PR[GP1:91,2] = PR[GP1:90,2] + 32.552;
   1:L PR[91] R[100]mm/sec CNT100;
   1:  PR[GP1:91,1] = PR[GP1:90,1] + -25.455;
   1:  PR[GP1:91,2] = PR[GP1:90,2] + 34.361;
   1:L PR[91] R[100]mm/sec CNT100;
   1:  PR[GP1:91,1] = PR[GP1:90,1] + -29.252;
   1:  PR[GP1:91,2] = PR[GP1:90,2] + 34.913;
   1:L PR[91] R[100]mm/sec CNT100;
   1:  PR[GP1:91,1] = PR[GP1:90,1] + -35.012;
   1:  PR[GP1:91,2] = PR[GP1:90,2] + 35.205;
   1:L PR[91] R[100]mm/sec CNT100;
   1:  PR[GP1:91,1] = PR[GP1:90,1] + -37.733;
   1:  PR[GP1:91,2] = PR[GP1:90,2] + 35.128;
   1:L PR[91] R[100]mm/sec CNT100;
   1:  PR[GP1:91,1] = PR[GP1:90,1] + -46.688;
   1:  PR[GP1:91,2] = PR[GP1:90,2] + 33.046;
   1:L PR[91] R[100]mm/sec CNT100;
   1:  PR[GP1:91,1] = PR[GP1:90,1] + -47.775;
   1:  PR[GP1:91,2] = PR[GP1:90,2] + 32.810;
   1:L PR[91] R[100]mm/sec CNT100;
   1:  PR[GP1:91,1] = PR[GP1:90,1] + -48.430;
   1:  PR[GP1:91,2] = PR[GP1:90,2] + 32.553;
   1:L PR[91] R[100]mm/sec CNT100;
   1:  PR[GP1:91,1] = PR[GP1:90,1] + -53.934;
   1:  PR[GP1:91,2] = PR[GP1:90,2] + 29.421;
   1:L PR[91] R[100]mm/sec CNT100;
   1:  PR[GP1:91,1] = PR[GP1:90,1] + -57.469;
   1:  PR[GP1:91,2] = PR[GP1:90,2] + 27.428;
   1:L PR[91] R[100]mm/sec CNT100;
   1:  PR[GP1:91,1] = PR[GP1:90,1] + -57.989;
   1:  PR[GP1:91,2] = PR[GP1:90,2] + 26.918;
   1:L PR[91] R[100]mm/sec CNT100;
   1:  PR[GP1:91,1] = PR[GP1:90,1] + -64.721;
   1:  PR[GP1:91,2] = PR[GP1:90,2] + 19.826;
   1:L PR[91] R[100]mm/sec CNT100;
   1:  PR[GP1:91,1] = PR[GP1:90,1] + -65.735;
   1:  PR[GP1:91,2] = PR[GP1:90,2] + 17.880;
   1:L PR[91] R[100]mm/sec CNT100;
   1:  PR[GP1:91,1] = PR[GP1:90,1] + -69.435;
   1:  PR[GP1:91,2] = PR[GP1:90,2] + 10.391;
   1:L PR[91] R[100]mm/sec CNT100;
   1:  PR[GP1:91,1] = PR[GP1:90,1] + -69.970;
   1:  PR[GP1:91,2] = PR[GP1:90,2] + 7.153;
   1:L PR[91] R[100]mm/sec CNT100;
   1:  PR[GP1:91,1] = PR[GP1:90,1] + -71.077;
   1:  PR[GP1:91,2] = PR[GP1:90,2] + -0.068;
   1:L PR[91] R[100]mm/sec CNT100;
   1:  PR[GP1:91,1] = PR[GP1:90,1] + -70.538;
   1:  PR[GP1:91,2] = PR[GP1:90,2] + -3.300;
   1:L PR[91] R[100]mm/sec CNT100;
   1:  PR[GP1:91,1] = PR[GP1:90,1] + -69.433;
   1:  PR[GP1:91,2] = PR[GP1:90,2] + -10.539;
   1:L PR[91] R[100]mm/sec CNT100;
   1:  PR[GP1:91,1] = PR[GP1:90,1] + -65.735;
   1:  PR[GP1:91,2] = PR[GP1:90,2] + -18.023;
   1:L PR[91] R[100]mm/sec CNT100;
   1:  PR[GP1:91,1] = PR[GP1:90,1] + -64.721;
   1:  PR[GP1:91,2] = PR[GP1:90,2] + -19.970;
   1:L PR[91] R[100]mm/sec CNT100;
   1:  PR[GP1:91,1] = PR[GP1:90,1] + -57.989;
   1:  PR[GP1:91,2] = PR[GP1:90,2] + -27.062;
   1:L PR[91] R[100]mm/sec CNT100;
   1:  PR[GP1:91,1] = PR[GP1:90,1] + -57.469;
   1:  PR[GP1:91,2] = PR[GP1:90,2] + -27.572;
   1:L PR[91] R[100]mm/sec CNT100;
   1:  PR[GP1:91,1] = PR[GP1:90,1] + -48.886;
   1:  PR[GP1:91,2] = PR[GP1:90,2] + -32.405;
   1:L PR[91] R[100]mm/sec CNT100;
   1:  PR[GP1:91,1] = PR[GP1:90,1] + -48.417;
   1:  PR[GP1:91,2] = PR[GP1:90,2] + -32.702;
   1:L PR[91] R[100]mm/sec CNT100;
   1:  PR[GP1:91,1] = PR[GP1:90,1] + -47.770;
   1:  PR[GP1:91,2] = PR[GP1:90,2] + -32.956;
   1:L PR[91] R[100]mm/sec CNT100;
   1:  PR[GP1:91,1] = PR[GP1:90,1] + -39.580;
   1:  PR[GP1:91,2] = PR[GP1:90,2] + -34.884;
   1:L PR[91] R[100]mm/sec CNT100;
   1:  PR[GP1:91,1] = PR[GP1:90,1] + -37.739;
   1:  PR[GP1:91,2] = PR[GP1:90,2] + -35.272;
   1:L PR[91] R[100]mm/sec CNT100;
   1:  PR[GP1:91,1] = PR[GP1:90,1] + -35.012;
   1:  PR[GP1:91,2] = PR[GP1:90,2] + -35.349;
   1:L PR[91] R[100]mm/sec CNT100;
   1:  PR[GP1:91,1] = PR[GP1:90,1] + -29.252;
   1:  PR[GP1:91,2] = PR[GP1:90,2] + -35.057;
   1:L PR[91] R[100]mm/sec CNT100;
   1:  PR[GP1:91,1] = PR[GP1:90,1] + -25.463;
   1:  PR[GP1:91,2] = PR[GP1:90,2] + -34.506;
   1:L PR[91] R[100]mm/sec CNT100;
   1:  PR[GP1:91,1] = PR[GP1:90,1] + -22.559;
   1:  PR[GP1:91,2] = PR[GP1:90,2] + -33.467;
   1:L PR[91] R[100]mm/sec CNT100;
   1:  PR[GP1:91,1] = PR[GP1:90,1] + -18.217;
   1:  PR[GP1:91,2] = PR[GP1:90,2] + -32.102;
   1:L PR[91] R[100]mm/sec CNT100;
   1:  PR[GP1:91,1] = PR[GP1:90,1] + -14.058;
   1:  PR[GP1:91,2] = PR[GP1:90,2] + -29.834;
   1:L PR[91] R[100]mm/sec CNT100;
   1:  PR[GP1:91,1] = PR[GP1:90,1] + -12.619;
   1:  PR[GP1:91,2] = PR[GP1:90,2] + -29.081;
   1:L PR[91] R[100]mm/sec CNT100;
   1:  PR[GP1:91,1] = PR[GP1:90,1] + -7.574;
   1:  PR[GP1:91,2] = PR[GP1:90,2] + -25.136;
   1:L PR[91] R[100]mm/sec CNT100;
   1:  PR[GP1:91,1] = PR[GP1:90,1] + -3.873;
   1:  PR[GP1:91,2] = PR[GP1:90,2] + -20.843;
   1:L PR[91] R[100]mm/sec CNT100;
   1:  PR[GP1:91,1] = PR[GP1:90,1] + -3.136;
   1:  PR[GP1:91,2] = PR[GP1:90,2] + -20.685;
   1:L PR[91] R[100]mm/sec CNT100;
   1:  PR[GP1:91,1] = PR[GP1:90,1] + 0.228;
   1:  PR[GP1:91,2] = PR[GP1:90,2] + -18.902;
   1:L PR[91] R[100]mm/sec CNT100;
   1:  PR[GP1:91,1] = PR[GP1:90,1] + 4.152;
   1:  PR[GP1:91,2] = PR[GP1:90,2] + -20.905;
   1:L PR[91] R[100]mm/sec CNT100;
   1:  PR[GP1:91,1] = PR[GP1:90,1] + 7.833;
   1:  PR[GP1:91,2] = PR[GP1:90,2] + -25.179;
   1:L PR[91] R[100]mm/sec CNT100;
   1:  PR[GP1:91,1] = PR[GP1:90,1] + 12.791;
   1:  PR[GP1:91,2] = PR[GP1:90,2] + -29.058;
   1:L PR[91] R[100]mm/sec CNT100;
   1:  PR[GP1:91,1] = PR[GP1:90,1] + 12.844;
   1:  PR[GP1:91,2] = PR[GP1:90,2] + -29.097;
   1:L PR[91] R[100]mm/sec CNT100;
   1:  PR[GP1:91,1] = PR[GP1:90,1] + 14.270;
   1:  PR[GP1:91,2] = PR[GP1:90,2] + -29.841;
   1:L PR[91] R[100]mm/sec CNT100;
   1:  PR[GP1:91,1] = PR[GP1:90,1] + 18.427;
   1:  PR[GP1:91,2] = PR[GP1:90,2] + -32.102;
   1:L PR[91] R[100]mm/sec CNT100;
   1:  PR[GP1:91,1] = PR[GP1:90,1] + 20.094;
   1:  PR[GP1:91,2] = PR[GP1:90,2] + -32.689;
   1:L PR[91] R[100]mm/sec CNT100;
   1:  PR[GP1:91,1] = PR[GP1:90,1] + 25.665;
   1:  PR[GP1:91,2] = PR[GP1:90,2] + -34.502;
   1:L PR[91] R[100]mm/sec CNT100;
   1:  PR[GP1:91,1] = PR[GP1:90,1] + 29.459;
   1:  PR[GP1:91,2] = PR[GP1:90,2] + -35.057;
   1:L PR[91] R[100]mm/sec CNT100;
   1:  PR[GP1:91,1] = PR[GP1:90,1] + 35.219;
   1:  PR[GP1:91,2] = PR[GP1:90,2] + -35.350;
   1:L PR[91] R[100]mm/sec CNT100;
   1:  PR[GP1:91,1] = PR[GP1:90,1] + 37.932;
   1:  PR[GP1:91,2] = PR[GP1:90,2] + -35.275;
   1:L PR[91] R[100]mm/sec CNT100;
   1:  PR[GP1:91,1] = PR[GP1:90,1] + 46.893;
   1:  PR[GP1:91,2] = PR[GP1:90,2] + -33.189;
   1:L PR[91] R[100]mm/sec CNT100;
   1:  PR[GP1:91,1] = PR[GP1:90,1] + 47.982;
   1:  PR[GP1:91,2] = PR[GP1:90,2] + -32.953;
   1:L PR[91] R[100]mm/sec CNT100;
   1:  PR[GP1:91,1] = PR[GP1:90,1] + 48.640;
   1:  PR[GP1:91,2] = PR[GP1:90,2] + -32.696;
   1:L PR[91] R[100]mm/sec CNT100;
   1:  PR[GP1:91,1] = PR[GP1:90,1] + 54.147;
   1:  PR[GP1:91,2] = PR[GP1:90,2] + -29.567;
   1:L PR[91] R[100]mm/sec CNT100;
   1:  PR[GP1:91,1] = PR[GP1:90,1] + 57.681;
   1:  PR[GP1:91,2] = PR[GP1:90,2] + -27.578;
   1:L PR[91] R[100]mm/sec CNT100;
   1:  PR[GP1:91,1] = PR[GP1:90,1] + 58.201;
   1:  PR[GP1:91,2] = PR[GP1:90,2] + -27.067;
   1:L PR[91] R[100]mm/sec CNT100;
   1:  PR[GP1:91,1] = PR[GP1:90,1] + 64.934;
   1:  PR[GP1:91,2] = PR[GP1:90,2] + -19.955;
   1:L PR[91] R[100]mm/sec CNT100;
   1:  PR[GP1:91,1] = PR[GP1:90,1] + 65.948;
   1:  PR[GP1:91,2] = PR[GP1:90,2] + -18.013;
   1:L PR[91] R[100]mm/sec CNT100;
   1:  PR[GP1:91,1] = PR[GP1:90,1] + 69.648;
   1:  PR[GP1:91,2] = PR[GP1:90,2] + -10.561;
   1:L PR[91] R[100]mm/sec CNT100;
   1:  PR[GP1:91,1] = PR[GP1:90,1] + 70.183;
   1:  PR[GP1:91,2] = PR[GP1:90,2] + -7.318;
   1:L PR[91] R[100]mm/sec CNT100;
   1:  PR[GP1:91,1] = PR[GP1:90,1] + 71.290;
   1:  PR[GP1:91,2] = PR[GP1:90,2] + -0.076;
   1:L PR[91] R[100]mm/sec CNT100;
   1:  PR[GP1:91,1] = PR[GP1:90,1] + 70.751;
   1:  PR[GP1:91,2] = PR[GP1:90,2] + 3.162;
   1:L PR[91] R[100]mm/sec CNT100;
   1:  PR[GP1:91,1] = PR[GP1:90,1] + 69.646;
   1:  PR[GP1:91,2] = PR[GP1:90,2] + 10.420;
   1:L PR[91] R[100]mm/sec CNT100;
   1:  PR[GP1:91,1] = PR[GP1:90,1] + 65.948;
   1:  PR[GP1:91,2] = PR[GP1:90,2] + 17.869;
   1:L PR[91] R[100]mm/sec CNT100;
   1:  PR[GP1:91,1] = PR[GP1:90,1] + 64.934;
   1:  PR[GP1:91,2] = PR[GP1:90,2] + 19.811;
   1:L PR[91] R[100]mm/sec CNT100;
   1:  PR[GP1:91,1] = PR[GP1:90,1] + 58.201;
   1:  PR[GP1:91,2] = PR[GP1:90,2] + 26.923;
   1:L PR[91] R[100]mm/sec CNT100;
   1:  PR[GP1:91,1] = PR[GP1:90,1] + 57.681;
   1:  PR[GP1:91,2] = PR[GP1:90,2] + 27.434;
   1:L PR[91] R[100]mm/sec CNT100;
   1:  PR[GP1:91,1] = PR[GP1:90,1] + 49.095;
   1:  PR[GP1:91,2] = PR[GP1:90,2] + 32.262;
   1:L PR[91] R[100]mm/sec CNT100;
   1:  PR[GP1:91,1] = PR[GP1:90,1] + 48.627;
   1:  PR[GP1:91,2] = PR[GP1:90,2] + 32.557;
   1:L PR[91] R[100]mm/sec CNT100;
   1:  PR[GP1:91,1] = PR[GP1:90,1] + 47.977;
   1:  PR[GP1:91,2] = PR[GP1:90,2] + 32.811;
   1:L PR[91] R[100]mm/sec CNT100;
   1:  PR[GP1:91,1] = PR[GP1:90,1] + 39.782;
   1:  PR[GP1:91,2] = PR[GP1:90,2] + 34.743;
   1:L PR[91] R[100]mm/sec CNT100;
   1:  PR[GP1:91,1] = PR[GP1:90,1] + 37.939;
   1:  PR[GP1:91,2] = PR[GP1:90,2] + 35.130;
   1:L PR[91] R[100]mm/sec CNT100;
   1:  PR[GP1:91,1] = PR[GP1:90,1] + 35.219;
   1:  PR[GP1:91,2] = PR[GP1:90,2] + 35.206;
   1:L PR[91] R[100]mm/sec CNT100;
   1:  PR[GP1:91,1] = PR[GP1:90,1] + 29.459;
   1:  PR[GP1:91,2] = PR[GP1:90,2] + 34.913;
   1:L PR[91] R[100]mm/sec CNT100;
   1:  PR[GP1:91,1] = PR[GP1:90,1] + 25.673;
   1:  PR[GP1:91,2] = PR[GP1:90,2] + 34.359;
   1:L PR[91] R[100]mm/sec CNT100;
   1:  PR[GP1:91,1] = PR[GP1:90,1] + 22.770;
   1:  PR[GP1:91,2] = PR[GP1:90,2] + 33.321;
   1:L PR[91] R[100]mm/sec CNT100;
   1:  PR[GP1:91,1] = PR[GP1:90,1] + 18.418;
   1:  PR[GP1:91,2] = PR[GP1:90,2] + 31.953;
   1:L PR[91] R[100]mm/sec CNT100;
   1:  PR[GP1:91,1] = PR[GP1:90,1] + 14.270;
   1:  PR[GP1:91,2] = PR[GP1:90,2] + 29.697;
   1:L PR[91] R[100]mm/sec CNT100;
   1:  PR[GP1:91,1] = PR[GP1:90,1] + 12.841;
   1:  PR[GP1:91,2] = PR[GP1:90,2] + 28.951;
   1:L PR[91] R[100]mm/sec CNT100;
   1:  PR[GP1:91,1] = PR[GP1:90,1] + 12.815;
   1:  PR[GP1:91,2] = PR[GP1:90,2] + 28.933;
   1:L PR[91] R[100]mm/sec CNT100;
   1:  PR[GP1:91,1] = PR[GP1:90,1] + 7.881;
   1:  PR[GP1:91,2] = PR[GP1:90,2] + 25.072;
   1:L PR[91] R[100]mm/sec CNT100;
   1:  PR[GP1:91,1] = PR[GP1:90,1] + 4.133;
   1:  PR[GP1:91,2] = PR[GP1:90,2] + 20.710;
   1:L PR[91] R[100]mm/sec CNT100;
   1:  PR[GP1:91,1] = PR[GP1:90,1] + 3.756;
   1:  PR[GP1:91,2] = PR[GP1:90,2] + 20.561;
   1:L PR[91] R[100]mm/sec CNT100;
   1:  PR[GP1:91,1] = PR[GP1:90,1] + 0.341;
   1:  PR[GP1:91,2] = PR[GP1:90,2] + 18.816;
   1:L PR[91] R[100]mm/sec CNT100;
   1:  ! -- Layer/Ebene 66 -- !;
   1:  PR[91] = PR[90];
   1:  PR[GP1:91,1] = PR[GP1:90,1] + -0.413;
   1:  PR[GP1:91,2] = PR[GP1:90,2] + 19.248;
   1:  PR[GP1:91,3] = PR[GP1:90,3] + 40.565;
   1:L PR[91] R[100]mm/sec CNT100;
   1:  PR[GP1:91,1] = PR[GP1:90,1] + -3.898;
   1:  PR[GP1:91,2] = PR[GP1:90,2] + 21.021;
   1:L PR[91] R[100]mm/sec CNT100;
   1:  PR[GP1:91,1] = PR[GP1:90,1] + -7.466;
   1:  PR[GP1:91,2] = PR[GP1:90,2] + 25.169;
   1:L PR[91] R[100]mm/sec CNT100;
   1:  PR[GP1:91,1] = PR[GP1:90,1] + -12.250;
   1:  PR[GP1:91,2] = PR[GP1:90,2] + 28.915;
   1:L PR[91] R[100]mm/sec CNT100;
   1:  PR[GP1:91,1] = PR[GP1:90,1] + -12.396;
   1:  PR[GP1:91,2] = PR[GP1:90,2] + 29.018;
   1:L PR[91] R[100]mm/sec CNT100;
   1:  PR[GP1:91,1] = PR[GP1:90,1] + -16.295;
   1:  PR[GP1:91,2] = PR[GP1:90,2] + 31.058;
   1:L PR[91] R[100]mm/sec CNT100;
   1:  PR[GP1:91,1] = PR[GP1:90,1] + -18.209;
   1:  PR[GP1:91,2] = PR[GP1:90,2] + 32.102;
   1:L PR[91] R[100]mm/sec CNT100;
   1:  PR[GP1:91,1] = PR[GP1:90,1] + -18.956;
   1:  PR[GP1:91,2] = PR[GP1:90,2] + 32.365;
   1:L PR[91] R[100]mm/sec CNT100;
   1:  PR[GP1:91,1] = PR[GP1:90,1] + -25.153;
   1:  PR[GP1:91,2] = PR[GP1:90,2] + 34.382;
   1:L PR[91] R[100]mm/sec CNT100;
   1:  PR[GP1:91,1] = PR[GP1:90,1] + -29.392;
   1:  PR[GP1:91,2] = PR[GP1:90,2] + 34.999;
   1:L PR[91] R[100]mm/sec CNT100;
   1:  PR[GP1:91,1] = PR[GP1:90,1] + -34.361;
   1:  PR[GP1:91,2] = PR[GP1:90,2] + 35.251;
   1:L PR[91] R[100]mm/sec CNT100;
   1:  PR[GP1:91,1] = PR[GP1:90,1] + -37.613;
   1:  PR[GP1:91,2] = PR[GP1:90,2] + 35.158;
   1:L PR[91] R[100]mm/sec CNT100;
   1:  PR[GP1:91,1] = PR[GP1:90,1] + -45.685;
   1:  PR[GP1:91,2] = PR[GP1:90,2] + 33.282;
   1:L PR[91] R[100]mm/sec CNT100;
   1:  PR[GP1:91,1] = PR[GP1:90,1] + -47.381;
   1:  PR[GP1:91,2] = PR[GP1:90,2] + 32.914;
   1:L PR[91] R[100]mm/sec CNT100;
   1:  PR[GP1:91,1] = PR[GP1:90,1] + -48.434;
   1:  PR[GP1:91,2] = PR[GP1:90,2] + 32.500;
   1:L PR[91] R[100]mm/sec CNT100;
   1:  PR[GP1:91,1] = PR[GP1:90,1] + -57.408;
   1:  PR[GP1:91,2] = PR[GP1:90,2] + 27.396;
   1:L PR[91] R[100]mm/sec CNT100;
   1:  PR[GP1:91,1] = PR[GP1:90,1] + -64.636;
   1:  PR[GP1:91,2] = PR[GP1:90,2] + 19.789;
   1:L PR[91] R[100]mm/sec CNT100;
   1:  PR[GP1:91,1] = PR[GP1:90,1] + -65.354;
   1:  PR[GP1:91,2] = PR[GP1:90,2] + 18.410;
   1:L PR[91] R[100]mm/sec CNT100;
   1:  PR[GP1:91,1] = PR[GP1:90,1] + -69.327;
   1:  PR[GP1:91,2] = PR[GP1:90,2] + 10.370;
   1:L PR[91] R[100]mm/sec CNT100;
   1:  PR[GP1:91,1] = PR[GP1:90,1] + -69.753;
   1:  PR[GP1:91,2] = PR[GP1:90,2] + 7.786;
   1:L PR[91] R[100]mm/sec CNT100;
   1:  PR[GP1:91,1] = PR[GP1:90,1] + -70.957;
   1:  PR[GP1:91,2] = PR[GP1:90,2] + -0.068;
   1:L PR[91] R[100]mm/sec CNT100;
   1:  PR[GP1:91,1] = PR[GP1:90,1] + -70.511;
   1:  PR[GP1:91,2] = PR[GP1:90,2] + -2.745;
   1:L PR[91] R[100]mm/sec CNT100;
   1:  PR[GP1:91,1] = PR[GP1:90,1] + -69.325;
   1:  PR[GP1:91,2] = PR[GP1:90,2] + -10.518;
   1:L PR[91] R[100]mm/sec CNT100;
   1:  PR[GP1:91,1] = PR[GP1:90,1] + -65.354;
   1:  PR[GP1:91,2] = PR[GP1:90,2] + -18.554;
   1:L PR[91] R[100]mm/sec CNT100;
   1:  PR[GP1:91,1] = PR[GP1:90,1] + -64.636;
   1:  PR[GP1:91,2] = PR[GP1:90,2] + -19.933;
   1:L PR[91] R[100]mm/sec CNT100;
   1:  PR[GP1:91,1] = PR[GP1:90,1] + -57.409;
   1:  PR[GP1:91,2] = PR[GP1:90,2] + -27.539;
   1:L PR[91] R[100]mm/sec CNT100;
   1:  PR[GP1:91,1] = PR[GP1:90,1] + -49.161;
   1:  PR[GP1:91,2] = PR[GP1:90,2] + -32.180;
   1:L PR[91] R[100]mm/sec CNT100;
   1:  PR[GP1:91,1] = PR[GP1:90,1] + -48.421;
   1:  PR[GP1:91,2] = PR[GP1:90,2] + -32.649;
   1:L PR[91] R[100]mm/sec CNT100;
   1:  PR[GP1:91,1] = PR[GP1:90,1] + -47.376;
   1:  PR[GP1:91,2] = PR[GP1:90,2] + -33.060;
   1:L PR[91] R[100]mm/sec CNT100;
   1:  PR[GP1:91,1] = PR[GP1:90,1] + -39.820;
   1:  PR[GP1:91,2] = PR[GP1:90,2] + -34.838;
   1:L PR[91] R[100]mm/sec CNT100;
   1:  PR[GP1:91,1] = PR[GP1:90,1] + -37.620;
   1:  PR[GP1:91,2] = PR[GP1:90,2] + -35.302;
   1:L PR[91] R[100]mm/sec CNT100;
   1:  PR[GP1:91,1] = PR[GP1:90,1] + -34.361;
   1:  PR[GP1:91,2] = PR[GP1:90,2] + -35.395;
   1:L PR[91] R[100]mm/sec CNT100;
   1:  PR[GP1:91,1] = PR[GP1:90,1] + -29.392;
   1:  PR[GP1:91,2] = PR[GP1:90,2] + -35.143;
   1:L PR[91] R[100]mm/sec CNT100;
   1:  PR[GP1:91,1] = PR[GP1:90,1] + -25.162;
   1:  PR[GP1:91,2] = PR[GP1:90,2] + -34.528;
   1:L PR[91] R[100]mm/sec CNT100;
   1:  PR[GP1:91,1] = PR[GP1:90,1] + -22.907;
   1:  PR[GP1:91,2] = PR[GP1:90,2] + -33.720;
   1:L PR[91] R[100]mm/sec CNT100;
   1:  PR[GP1:91,1] = PR[GP1:90,1] + -18.200;
   1:  PR[GP1:91,2] = PR[GP1:90,2] + -32.241;
   1:L PR[91] R[100]mm/sec CNT100;
   1:  PR[GP1:91,1] = PR[GP1:90,1] + -16.295;
   1:  PR[GP1:91,2] = PR[GP1:90,2] + -31.202;
   1:L PR[91] R[100]mm/sec CNT100;
   1:  PR[GP1:91,1] = PR[GP1:90,1] + -12.399;
   1:  PR[GP1:91,2] = PR[GP1:90,2] + -29.164;
   1:L PR[91] R[100]mm/sec CNT100;
   1:  PR[GP1:91,1] = PR[GP1:90,1] + -12.181;
   1:  PR[GP1:91,2] = PR[GP1:90,2] + -29.005;
   1:L PR[91] R[100]mm/sec CNT100;
   1:  PR[GP1:91,1] = PR[GP1:90,1] + -7.401;
   1:  PR[GP1:91,2] = PR[GP1:90,2] + -25.262;
   1:L PR[91] R[100]mm/sec CNT100;
   1:  PR[GP1:91,1] = PR[GP1:90,1] + -3.843;
   1:  PR[GP1:91,2] = PR[GP1:90,2] + -21.136;
   1:L PR[91] R[100]mm/sec CNT100;
   1:  PR[GP1:91,1] = PR[GP1:90,1] + -2.969;
   1:  PR[GP1:91,2] = PR[GP1:90,2] + -20.948;
   1:L PR[91] R[100]mm/sec CNT100;
   1:  PR[GP1:91,1] = PR[GP1:90,1] + 0.269;
   1:  PR[GP1:91,2] = PR[GP1:90,2] + -19.232;
   1:L PR[91] R[100]mm/sec CNT100;
   1:  PR[GP1:91,1] = PR[GP1:90,1] + 4.122;
   1:  PR[GP1:91,2] = PR[GP1:90,2] + -21.198;
   1:L PR[91] R[100]mm/sec CNT100;
   1:  PR[GP1:91,1] = PR[GP1:90,1] + 7.657;
   1:  PR[GP1:91,2] = PR[GP1:90,2] + -25.303;
   1:L PR[91] R[100]mm/sec CNT100;
   1:  PR[GP1:91,1] = PR[GP1:90,1] + 12.416;
   1:  PR[GP1:91,2] = PR[GP1:90,2] + -29.026;
   1:L PR[91] R[100]mm/sec CNT100;
   1:  PR[GP1:91,1] = PR[GP1:90,1] + 12.633;
   1:  PR[GP1:91,2] = PR[GP1:90,2] + -29.184;
   1:L PR[91] R[100]mm/sec CNT100;
   1:  PR[GP1:91,1] = PR[GP1:90,1] + 16.507;
   1:  PR[GP1:91,2] = PR[GP1:90,2] + -31.206;
   1:L PR[91] R[100]mm/sec CNT100;
   1:  PR[GP1:91,1] = PR[GP1:90,1] + 18.409;
   1:  PR[GP1:91,2] = PR[GP1:90,2] + -32.240;
   1:L PR[91] R[100]mm/sec CNT100;
   1:  PR[GP1:91,1] = PR[GP1:90,1] + 19.152;
   1:  PR[GP1:91,2] = PR[GP1:90,2] + -32.502;
   1:L PR[91] R[100]mm/sec CNT100;
   1:  PR[GP1:91,1] = PR[GP1:90,1] + 25.363;
   1:  PR[GP1:91,2] = PR[GP1:90,2] + -34.523;
   1:L PR[91] R[100]mm/sec CNT100;
   1:  PR[GP1:91,1] = PR[GP1:90,1] + 29.598;
   1:  PR[GP1:91,2] = PR[GP1:90,2] + -35.142;
   1:L PR[91] R[100]mm/sec CNT100;
   1:  PR[GP1:91,1] = PR[GP1:90,1] + 34.567;
   1:  PR[GP1:91,2] = PR[GP1:90,2] + -35.395;
   1:L PR[91] R[100]mm/sec CNT100;
   1:  PR[GP1:91,1] = PR[GP1:90,1] + 37.810;
   1:  PR[GP1:91,2] = PR[GP1:90,2] + -35.305;
   1:L PR[91] R[100]mm/sec CNT100;
   1:  PR[GP1:91,1] = PR[GP1:90,1] + 45.885;
   1:  PR[GP1:91,2] = PR[GP1:90,2] + -33.425;
   1:L PR[91] R[100]mm/sec CNT100;
   1:  PR[GP1:91,1] = PR[GP1:90,1] + 47.584;
   1:  PR[GP1:91,2] = PR[GP1:90,2] + -33.058;
   1:L PR[91] R[100]mm/sec CNT100;
   1:  PR[GP1:91,1] = PR[GP1:90,1] + 48.643;
   1:  PR[GP1:91,2] = PR[GP1:90,2] + -32.644;
   1:L PR[91] R[100]mm/sec CNT100;
   1:  PR[GP1:91,1] = PR[GP1:90,1] + 57.621;
   1:  PR[GP1:91,2] = PR[GP1:90,2] + -27.546;
   1:L PR[91] R[100]mm/sec CNT100;
   1:  PR[GP1:91,1] = PR[GP1:90,1] + 64.848;
   1:  PR[GP1:91,2] = PR[GP1:90,2] + -19.918;
   1:L PR[91] R[100]mm/sec CNT100;
   1:  PR[GP1:91,1] = PR[GP1:90,1] + 65.567;
   1:  PR[GP1:91,2] = PR[GP1:90,2] + -18.541;
   1:L PR[91] R[100]mm/sec CNT100;
   1:  PR[GP1:91,1] = PR[GP1:90,1] + 69.540;
   1:  PR[GP1:91,2] = PR[GP1:90,2] + -10.541;
   1:L PR[91] R[100]mm/sec CNT100;
   1:  PR[GP1:91,1] = PR[GP1:90,1] + 69.966;
   1:  PR[GP1:91,2] = PR[GP1:90,2] + -7.953;
   1:L PR[91] R[100]mm/sec CNT100;
   1:  PR[GP1:91,1] = PR[GP1:90,1] + 71.171;
   1:  PR[GP1:91,2] = PR[GP1:90,2] + -0.076;
   1:L PR[91] R[100]mm/sec CNT100;
   1:  PR[GP1:91,1] = PR[GP1:90,1] + 70.724;
   1:  PR[GP1:91,2] = PR[GP1:90,2] + 2.606;
   1:L PR[91] R[100]mm/sec CNT100;
   1:  PR[GP1:91,1] = PR[GP1:90,1] + 69.538;
   1:  PR[GP1:91,2] = PR[GP1:90,2] + 10.400;
   1:L PR[91] R[100]mm/sec CNT100;
   1:  PR[GP1:91,1] = PR[GP1:90,1] + 65.567;
   1:  PR[GP1:91,2] = PR[GP1:90,2] + 18.397;
   1:L PR[91] R[100]mm/sec CNT100;
   1:  PR[GP1:91,1] = PR[GP1:90,1] + 64.848;
   1:  PR[GP1:91,2] = PR[GP1:90,2] + 19.774;
   1:L PR[91] R[100]mm/sec CNT100;
   1:  PR[GP1:91,1] = PR[GP1:90,1] + 57.622;
   1:  PR[GP1:91,2] = PR[GP1:90,2] + 27.401;
   1:L PR[91] R[100]mm/sec CNT100;
   1:  PR[GP1:91,1] = PR[GP1:90,1] + 49.368;
   1:  PR[GP1:91,2] = PR[GP1:90,2] + 32.039;
   1:L PR[91] R[100]mm/sec CNT100;
   1:  PR[GP1:91,1] = PR[GP1:90,1] + 48.630;
   1:  PR[GP1:91,2] = PR[GP1:90,2] + 32.505;
   1:L PR[91] R[100]mm/sec CNT100;
   1:  PR[GP1:91,1] = PR[GP1:90,1] + 47.579;
   1:  PR[GP1:91,2] = PR[GP1:90,2] + 32.916;
   1:L PR[91] R[100]mm/sec CNT100;
   1:  PR[GP1:91,1] = PR[GP1:90,1] + 40.020;
   1:  PR[GP1:91,2] = PR[GP1:90,2] + 34.698;
   1:L PR[91] R[100]mm/sec CNT100;
   1:  PR[GP1:91,1] = PR[GP1:90,1] + 37.816;
   1:  PR[GP1:91,2] = PR[GP1:90,2] + 35.161;
   1:L PR[91] R[100]mm/sec CNT100;
   1:  PR[GP1:91,1] = PR[GP1:90,1] + 34.567;
   1:  PR[GP1:91,2] = PR[GP1:90,2] + 35.251;
   1:L PR[91] R[100]mm/sec CNT100;
   1:  PR[GP1:91,1] = PR[GP1:90,1] + 29.598;
   1:  PR[GP1:91,2] = PR[GP1:90,2] + 34.998;
   1:L PR[91] R[100]mm/sec CNT100;
   1:  PR[GP1:91,1] = PR[GP1:90,1] + 25.371;
   1:  PR[GP1:91,2] = PR[GP1:90,2] + 34.380;
   1:L PR[91] R[100]mm/sec CNT100;
   1:  PR[GP1:91,1] = PR[GP1:90,1] + 23.117;
   1:  PR[GP1:91,2] = PR[GP1:90,2] + 33.574;
   1:L PR[91] R[100]mm/sec CNT100;
   1:  PR[GP1:91,1] = PR[GP1:90,1] + 18.400;
   1:  PR[GP1:91,2] = PR[GP1:90,2] + 32.091;
   1:L PR[91] R[100]mm/sec CNT100;
   1:  PR[GP1:91,1] = PR[GP1:90,1] + 16.508;
   1:  PR[GP1:91,2] = PR[GP1:90,2] + 31.062;
   1:L PR[91] R[100]mm/sec CNT100;
   1:  PR[GP1:91,1] = PR[GP1:90,1] + 12.629;
   1:  PR[GP1:91,2] = PR[GP1:90,2] + 29.038;
   1:L PR[91] R[100]mm/sec CNT100;
   1:  PR[GP1:91,1] = PR[GP1:90,1] + 12.484;
   1:  PR[GP1:91,2] = PR[GP1:90,2] + 28.935;
   1:L PR[91] R[100]mm/sec CNT100;
   1:  PR[GP1:91,1] = PR[GP1:90,1] + 7.723;
   1:  PR[GP1:91,2] = PR[GP1:90,2] + 25.210;
   1:L PR[91] R[100]mm/sec CNT100;
   1:  PR[GP1:91,1] = PR[GP1:90,1] + 4.103;
   1:  PR[GP1:91,2] = PR[GP1:90,2] + 20.997;
   1:L PR[91] R[100]mm/sec CNT100;
   1:  PR[GP1:91,1] = PR[GP1:90,1] + 3.667;
   1:  PR[GP1:91,2] = PR[GP1:90,2] + 20.825;
   1:L PR[91] R[100]mm/sec CNT100;
   1:  PR[GP1:91,1] = PR[GP1:90,1] + 0.382;
   1:  PR[GP1:91,2] = PR[GP1:90,2] + 19.145;
   1:L PR[91] R[100]mm/sec CNT100;
   1:  ! -- Layer/Ebene 67 -- !;
   1:  PR[91] = PR[90];
   1:  PR[GP1:91,1] = PR[GP1:90,1] + -0.502;
   1:  PR[GP1:91,2] = PR[GP1:90,2] + 19.594;
   1:  PR[GP1:91,3] = PR[GP1:90,3] + 41.175;
   1:L PR[91] R[100]mm/sec CNT100;
   1:  PR[GP1:91,1] = PR[GP1:90,1] + -3.869;
   1:  PR[GP1:91,2] = PR[GP1:90,2] + 21.307;
   1:L PR[91] R[100]mm/sec CNT100;
   1:  PR[GP1:91,1] = PR[GP1:90,1] + -7.310;
   1:  PR[GP1:91,2] = PR[GP1:90,2] + 25.308;
   1:L PR[91] R[100]mm/sec CNT100;
   1:  PR[GP1:91,1] = PR[GP1:90,1] + -11.920;
   1:  PR[GP1:91,2] = PR[GP1:90,2] + 28.918;
   1:L PR[91] R[100]mm/sec CNT100;
   1:  PR[GP1:91,1] = PR[GP1:90,1] + -12.185;
   1:  PR[GP1:91,2] = PR[GP1:90,2] + 29.106;
   1:L PR[91] R[100]mm/sec CNT100;
   1:  PR[GP1:91,1] = PR[GP1:90,1] + -18.137;
   1:  PR[GP1:91,2] = PR[GP1:90,2] + 32.220;
   1:L PR[91] R[100]mm/sec CNT100;
   1:  PR[GP1:91,1] = PR[GP1:90,1] + -24.852;
   1:  PR[GP1:91,2] = PR[GP1:90,2] + 34.403;
   1:L PR[91] R[100]mm/sec CNT100;
   1:  PR[GP1:91,1] = PR[GP1:90,1] + -29.531;
   1:  PR[GP1:91,2] = PR[GP1:90,2] + 35.084;
   1:L PR[91] R[100]mm/sec CNT100;
   1:  PR[GP1:91,1] = PR[GP1:90,1] + -33.711;
   1:  PR[GP1:91,2] = PR[GP1:90,2] + 35.296;
   1:L PR[91] R[100]mm/sec CNT100;
   1:  PR[GP1:91,1] = PR[GP1:90,1] + -37.494;
   1:  PR[GP1:91,2] = PR[GP1:90,2] + 35.189;
   1:L PR[91] R[100]mm/sec CNT100;
   1:  PR[GP1:91,1] = PR[GP1:90,1] + -44.682;
   1:  PR[GP1:91,2] = PR[GP1:90,2] + 33.517;
   1:L PR[91] R[100]mm/sec CNT100;
   1:  PR[GP1:91,1] = PR[GP1:90,1] + -46.987;
   1:  PR[GP1:91,2] = PR[GP1:90,2] + 33.018;
   1:L PR[91] R[100]mm/sec CNT100;
   1:  PR[GP1:91,1] = PR[GP1:90,1] + -48.438;
   1:  PR[GP1:91,2] = PR[GP1:90,2] + 32.446;
   1:L PR[91] R[100]mm/sec CNT100;
   1:  PR[GP1:91,1] = PR[GP1:90,1] + -56.958;
   1:  PR[GP1:91,2] = PR[GP1:90,2] + 27.599;
   1:L PR[91] R[100]mm/sec CNT100;
   1:  PR[GP1:91,1] = PR[GP1:90,1] + -57.238;
   1:  PR[GP1:91,2] = PR[GP1:90,2] + 27.425;
   1:L PR[91] R[100]mm/sec CNT100;
   1:  PR[GP1:91,1] = PR[GP1:90,1] + -57.400;
   1:  PR[GP1:91,2] = PR[GP1:90,2] + 27.280;
   1:L PR[91] R[100]mm/sec CNT100;
   1:  PR[GP1:91,1] = PR[GP1:90,1] + -64.551;
   1:  PR[GP1:91,2] = PR[GP1:90,2] + 19.753;
   1:L PR[91] R[100]mm/sec CNT100;
   1:  PR[GP1:91,1] = PR[GP1:90,1] + -64.973;
   1:  PR[GP1:91,2] = PR[GP1:90,2] + 18.941;
   1:L PR[91] R[100]mm/sec CNT100;
   1:  PR[GP1:91,1] = PR[GP1:90,1] + -69.218;
   1:  PR[GP1:91,2] = PR[GP1:90,2] + 10.349;
   1:L PR[91] R[100]mm/sec CNT100;
   1:  PR[GP1:91,1] = PR[GP1:90,1] + -69.537;
   1:  PR[GP1:91,2] = PR[GP1:90,2] + 8.419;
   1:L PR[91] R[100]mm/sec CNT100;
   1:  PR[GP1:91,1] = PR[GP1:90,1] + -70.838;
   1:  PR[GP1:91,2] = PR[GP1:90,2] + -0.068;
   1:L PR[91] R[100]mm/sec CNT100;
   1:  PR[GP1:91,1] = PR[GP1:90,1] + -70.484;
   1:  PR[GP1:91,2] = PR[GP1:90,2] + -2.191;
   1:L PR[91] R[100]mm/sec CNT100;
   1:  PR[GP1:91,1] = PR[GP1:90,1] + -69.217;
   1:  PR[GP1:91,2] = PR[GP1:90,2] + -10.497;
   1:L PR[91] R[100]mm/sec CNT100;
   1:  PR[GP1:91,1] = PR[GP1:90,1] + -64.974;
   1:  PR[GP1:91,2] = PR[GP1:90,2] + -19.085;
   1:L PR[91] R[100]mm/sec CNT100;
   1:  PR[GP1:91,1] = PR[GP1:90,1] + -64.551;
   1:  PR[GP1:91,2] = PR[GP1:90,2] + -19.897;
   1:L PR[91] R[100]mm/sec CNT100;
   1:  PR[GP1:91,1] = PR[GP1:90,1] + -57.400;
   1:  PR[GP1:91,2] = PR[GP1:90,2] + -27.424;
   1:L PR[91] R[100]mm/sec CNT100;
   1:  PR[GP1:91,1] = PR[GP1:90,1] + -57.248;
   1:  PR[GP1:91,2] = PR[GP1:90,2] + -27.561;
   1:L PR[91] R[100]mm/sec CNT100;
   1:  PR[GP1:91,1] = PR[GP1:90,1] + -49.437;
   1:  PR[GP1:91,2] = PR[GP1:90,2] + -31.954;
   1:L PR[91] R[100]mm/sec CNT100;
   1:  PR[GP1:91,1] = PR[GP1:90,1] + -48.425;
   1:  PR[GP1:91,2] = PR[GP1:90,2] + -32.596;
   1:L PR[91] R[100]mm/sec CNT100;
   1:  PR[GP1:91,1] = PR[GP1:90,1] + -46.981;
   1:  PR[GP1:91,2] = PR[GP1:90,2] + -33.164;
   1:L PR[91] R[100]mm/sec CNT100;
   1:  PR[GP1:91,1] = PR[GP1:90,1] + -40.060;
   1:  PR[GP1:91,2] = PR[GP1:90,2] + -34.793;
   1:L PR[91] R[100]mm/sec CNT100;
   1:  PR[GP1:91,1] = PR[GP1:90,1] + -37.500;
   1:  PR[GP1:91,2] = PR[GP1:90,2] + -35.332;
   1:L PR[91] R[100]mm/sec CNT100;
   1:  PR[GP1:91,1] = PR[GP1:90,1] + -33.711;
   1:  PR[GP1:91,2] = PR[GP1:90,2] + -35.440;
   1:L PR[91] R[100]mm/sec CNT100;
   1:  PR[GP1:91,1] = PR[GP1:90,1] + -29.531;
   1:  PR[GP1:91,2] = PR[GP1:90,2] + -35.228;
   1:L PR[91] R[100]mm/sec CNT100;
   1:  PR[GP1:91,1] = PR[GP1:90,1] + -24.861;
   1:  PR[GP1:91,2] = PR[GP1:90,2] + -34.549;
   1:L PR[91] R[100]mm/sec CNT100;
   1:  PR[GP1:91,1] = PR[GP1:90,1] + -23.254;
   1:  PR[GP1:91,2] = PR[GP1:90,2] + -33.974;
   1:L PR[91] R[100]mm/sec CNT100;
   1:  PR[GP1:91,1] = PR[GP1:90,1] + -18.134;
   1:  PR[GP1:91,2] = PR[GP1:90,2] + -32.362;
   1:L PR[91] R[100]mm/sec CNT100;
   1:  PR[GP1:91,1] = PR[GP1:90,1] + -12.188;
   1:  PR[GP1:91,2] = PR[GP1:90,2] + -29.251;
   1:L PR[91] R[100]mm/sec CNT100;
   1:  PR[GP1:91,1] = PR[GP1:90,1] + -11.807;
   1:  PR[GP1:91,2] = PR[GP1:90,2] + -28.974;
   1:L PR[91] R[100]mm/sec CNT100;
   1:  PR[GP1:91,1] = PR[GP1:90,1] + -7.227;
   1:  PR[GP1:91,2] = PR[GP1:90,2] + -25.388;
   1:L PR[91] R[100]mm/sec CNT100;
   1:  PR[GP1:91,1] = PR[GP1:90,1] + -3.814;
   1:  PR[GP1:91,2] = PR[GP1:90,2] + -21.429;
   1:L PR[91] R[100]mm/sec CNT100;
   1:  PR[GP1:91,1] = PR[GP1:90,1] + -2.803;
   1:  PR[GP1:91,2] = PR[GP1:90,2] + -21.212;
   1:L PR[91] R[100]mm/sec CNT100;
   1:  PR[GP1:91,1] = PR[GP1:90,1] + 0.310;
   1:  PR[GP1:91,2] = PR[GP1:90,2] + -19.562;
   1:L PR[91] R[100]mm/sec CNT100;
   1:  PR[GP1:91,1] = PR[GP1:90,1] + 4.092;
   1:  PR[GP1:91,2] = PR[GP1:90,2] + -21.491;
   1:L PR[91] R[100]mm/sec CNT100;
   1:  PR[GP1:91,1] = PR[GP1:90,1] + 7.482;
   1:  PR[GP1:91,2] = PR[GP1:90,2] + -25.427;
   1:L PR[91] R[100]mm/sec CNT100;
   1:  PR[GP1:91,1] = PR[GP1:90,1] + 12.041;
   1:  PR[GP1:91,2] = PR[GP1:90,2] + -28.994;
   1:L PR[91] R[100]mm/sec CNT100;
   1:  PR[GP1:91,1] = PR[GP1:90,1] + 12.421;
   1:  PR[GP1:91,2] = PR[GP1:90,2] + -29.270;
   1:L PR[91] R[100]mm/sec CNT100;
   1:  PR[GP1:91,1] = PR[GP1:90,1] + 18.334;
   1:  PR[GP1:91,2] = PR[GP1:90,2] + -32.356;
   1:L PR[91] R[100]mm/sec CNT100;
   1:  PR[GP1:91,1] = PR[GP1:90,1] + 25.061;
   1:  PR[GP1:91,2] = PR[GP1:90,2] + -34.544;
   1:L PR[91] R[100]mm/sec CNT100;
   1:  PR[GP1:91,1] = PR[GP1:90,1] + 29.737;
   1:  PR[GP1:91,2] = PR[GP1:90,2] + -35.228;
   1:L PR[91] R[100]mm/sec CNT100;
   1:  PR[GP1:91,1] = PR[GP1:90,1] + 33.914;
   1:  PR[GP1:91,2] = PR[GP1:90,2] + -35.440;
   1:L PR[91] R[100]mm/sec CNT100;
   1:  PR[GP1:91,1] = PR[GP1:90,1] + 37.687;
   1:  PR[GP1:91,2] = PR[GP1:90,2] + -35.336;
   1:L PR[91] R[100]mm/sec CNT100;
   1:  PR[GP1:91,1] = PR[GP1:90,1] + 44.877;
   1:  PR[GP1:91,2] = PR[GP1:90,2] + -33.662;
   1:L PR[91] R[100]mm/sec CNT100;
   1:  PR[GP1:91,1] = PR[GP1:90,1] + 47.187;
   1:  PR[GP1:91,2] = PR[GP1:90,2] + -33.162;
   1:L PR[91] R[100]mm/sec CNT100;
   1:  PR[GP1:91,1] = PR[GP1:90,1] + 48.645;
   1:  PR[GP1:91,2] = PR[GP1:90,2] + -32.592;
   1:L PR[91] R[100]mm/sec CNT100;
   1:  PR[GP1:91,1] = PR[GP1:90,1] + 57.169;
   1:  PR[GP1:91,2] = PR[GP1:90,2] + -27.749;
   1:L PR[91] R[100]mm/sec CNT100;
   1:  PR[GP1:91,1] = PR[GP1:90,1] + 57.449;
   1:  PR[GP1:91,2] = PR[GP1:90,2] + -27.577;
   1:L PR[91] R[100]mm/sec CNT100;
   1:  PR[GP1:91,1] = PR[GP1:90,1] + 57.609;
   1:  PR[GP1:91,2] = PR[GP1:90,2] + -27.433;
   1:L PR[91] R[100]mm/sec CNT100;
   1:  PR[GP1:91,1] = PR[GP1:90,1] + 64.763;
   1:  PR[GP1:91,2] = PR[GP1:90,2] + -19.880;
   1:L PR[91] R[100]mm/sec CNT100;
   1:  PR[GP1:91,1] = PR[GP1:90,1] + 65.186;
   1:  PR[GP1:91,2] = PR[GP1:90,2] + -19.070;
   1:L PR[91] R[100]mm/sec CNT100;
   1:  PR[GP1:91,1] = PR[GP1:90,1] + 69.431;
   1:  PR[GP1:91,2] = PR[GP1:90,2] + -10.520;
   1:L PR[91] R[100]mm/sec CNT100;
   1:  PR[GP1:91,1] = PR[GP1:90,1] + 69.750;
   1:  PR[GP1:91,2] = PR[GP1:90,2] + -8.587;
   1:L PR[91] R[100]mm/sec CNT100;
   1:  PR[GP1:91,1] = PR[GP1:90,1] + 71.051;
   1:  PR[GP1:91,2] = PR[GP1:90,2] + -0.076;
   1:L PR[91] R[100]mm/sec CNT100;
   1:  PR[GP1:91,1] = PR[GP1:90,1] + 70.697;
   1:  PR[GP1:91,2] = PR[GP1:90,2] + 2.051;
   1:L PR[91] R[100]mm/sec CNT100;
   1:  PR[GP1:91,1] = PR[GP1:90,1] + 69.430;
   1:  PR[GP1:91,2] = PR[GP1:90,2] + 10.380;
   1:L PR[91] R[100]mm/sec CNT100;
   1:  PR[GP1:91,1] = PR[GP1:90,1] + 65.187;
   1:  PR[GP1:91,2] = PR[GP1:90,2] + 18.926;
   1:L PR[91] R[100]mm/sec CNT100;
   1:  PR[GP1:91,1] = PR[GP1:90,1] + 64.763;
   1:  PR[GP1:91,2] = PR[GP1:90,2] + 19.736;
   1:L PR[91] R[100]mm/sec CNT100;
   1:  PR[GP1:91,1] = PR[GP1:90,1] + 57.609;
   1:  PR[GP1:91,2] = PR[GP1:90,2] + 27.289;
   1:L PR[91] R[100]mm/sec CNT100;
   1:  PR[GP1:91,1] = PR[GP1:90,1] + 57.458;
   1:  PR[GP1:91,2] = PR[GP1:90,2] + 27.425;
   1:L PR[91] R[100]mm/sec CNT100;
   1:  PR[GP1:91,1] = PR[GP1:90,1] + 49.641;
   1:  PR[GP1:91,2] = PR[GP1:90,2] + 31.817;
   1:L PR[91] R[100]mm/sec CNT100;
   1:  PR[GP1:91,1] = PR[GP1:90,1] + 48.632;
   1:  PR[GP1:91,2] = PR[GP1:90,2] + 32.453;
   1:L PR[91] R[100]mm/sec CNT100;
   1:  PR[GP1:91,1] = PR[GP1:90,1] + 47.181;
   1:  PR[GP1:91,2] = PR[GP1:90,2] + 33.021;
   1:L PR[91] R[100]mm/sec CNT100;
   1:  PR[GP1:91,1] = PR[GP1:90,1] + 40.257;
   1:  PR[GP1:91,2] = PR[GP1:90,2] + 34.653;
   1:L PR[91] R[100]mm/sec CNT100;
   1:  PR[GP1:91,1] = PR[GP1:90,1] + 37.694;
   1:  PR[GP1:91,2] = PR[GP1:90,2] + 35.191;
   1:L PR[91] R[100]mm/sec CNT100;
   1:  PR[GP1:91,1] = PR[GP1:90,1] + 33.914;
   1:  PR[GP1:91,2] = PR[GP1:90,2] + 35.296;
   1:L PR[91] R[100]mm/sec CNT100;
   1:  PR[GP1:91,1] = PR[GP1:90,1] + 29.737;
   1:  PR[GP1:91,2] = PR[GP1:90,2] + 35.084;
   1:L PR[91] R[100]mm/sec CNT100;
   1:  PR[GP1:91,1] = PR[GP1:90,1] + 25.069;
   1:  PR[GP1:91,2] = PR[GP1:90,2] + 34.401;
   1:L PR[91] R[100]mm/sec CNT100;
   1:  PR[GP1:91,1] = PR[GP1:90,1] + 23.464;
   1:  PR[GP1:91,2] = PR[GP1:90,2] + 33.827;
   1:L PR[91] R[100]mm/sec CNT100;
   1:  PR[GP1:91,1] = PR[GP1:90,1] + 18.332;
   1:  PR[GP1:91,2] = PR[GP1:90,2] + 32.211;
   1:L PR[91] R[100]mm/sec CNT100;
   1:  PR[GP1:91,1] = PR[GP1:90,1] + 12.418;
   1:  PR[GP1:91,2] = PR[GP1:90,2] + 29.125;
   1:L PR[91] R[100]mm/sec CNT100;
   1:  PR[GP1:91,1] = PR[GP1:90,1] + 12.153;
   1:  PR[GP1:91,2] = PR[GP1:90,2] + 28.938;
   1:L PR[91] R[100]mm/sec CNT100;
   1:  PR[GP1:91,1] = PR[GP1:90,1] + 7.566;
   1:  PR[GP1:91,2] = PR[GP1:90,2] + 25.348;
   1:L PR[91] R[100]mm/sec CNT100;
   1:  PR[GP1:91,1] = PR[GP1:90,1] + 4.073;
   1:  PR[GP1:91,2] = PR[GP1:90,2] + 21.283;
   1:L PR[91] R[100]mm/sec CNT100;
   1:  PR[GP1:91,1] = PR[GP1:90,1] + 3.579;
   1:  PR[GP1:91,2] = PR[GP1:90,2] + 21.088;
   1:L PR[91] R[100]mm/sec CNT100;
   1:  PR[GP1:91,1] = PR[GP1:90,1] + 0.423;
   1:  PR[GP1:91,2] = PR[GP1:90,2] + 19.475;
   1:L PR[91] R[100]mm/sec CNT100;
   1:  ! -- Layer/Ebene 68 -- !;
   1:  PR[91] = PR[90];
   1:  PR[GP1:91,1] = PR[GP1:90,1] + -0.591;
   1:  PR[GP1:91,2] = PR[GP1:90,2] + 19.941;
   1:  PR[GP1:91,3] = PR[GP1:90,3] + 41.785;
   1:L PR[91] R[100]mm/sec CNT100;
   1:  PR[GP1:91,1] = PR[GP1:90,1] + -3.840;
   1:  PR[GP1:91,2] = PR[GP1:90,2] + 21.594;
   1:L PR[91] R[100]mm/sec CNT100;
   1:  PR[GP1:91,1] = PR[GP1:90,1] + -7.154;
   1:  PR[GP1:91,2] = PR[GP1:90,2] + 25.447;
   1:L PR[91] R[100]mm/sec CNT100;
   1:  PR[GP1:91,1] = PR[GP1:90,1] + -11.590;
   1:  PR[GP1:91,2] = PR[GP1:90,2] + 28.922;
   1:L PR[91] R[100]mm/sec CNT100;
   1:  PR[GP1:91,1] = PR[GP1:90,1] + -11.974;
   1:  PR[GP1:91,2] = PR[GP1:90,2] + 29.193;
   1:L PR[91] R[100]mm/sec CNT100;
   1:  PR[GP1:91,1] = PR[GP1:90,1] + -17.795;
   1:  PR[GP1:91,2] = PR[GP1:90,2] + 32.238;
   1:L PR[91] R[100]mm/sec CNT100;
   1:  PR[GP1:91,1] = PR[GP1:90,1] + -24.550;
   1:  PR[GP1:91,2] = PR[GP1:90,2] + 34.425;
   1:L PR[91] R[100]mm/sec CNT100;
   1:  PR[GP1:91,1] = PR[GP1:90,1] + -29.671;
   1:  PR[GP1:91,2] = PR[GP1:90,2] + 35.170;
   1:L PR[91] R[100]mm/sec CNT100;
   1:  PR[GP1:91,1] = PR[GP1:90,1] + -33.060;
   1:  PR[GP1:91,2] = PR[GP1:90,2] + 35.341;
   1:L PR[91] R[100]mm/sec CNT100;
   1:  PR[GP1:91,1] = PR[GP1:90,1] + -37.374;
   1:  PR[GP1:91,2] = PR[GP1:90,2] + 35.219;
   1:L PR[91] R[100]mm/sec CNT100;
   1:  PR[GP1:91,1] = PR[GP1:90,1] + -43.679;
   1:  PR[GP1:91,2] = PR[GP1:90,2] + 33.753;
   1:L PR[91] R[100]mm/sec CNT100;
   1:  PR[GP1:91,1] = PR[GP1:90,1] + -46.592;
   1:  PR[GP1:91,2] = PR[GP1:90,2] + 33.122;
   1:L PR[91] R[100]mm/sec CNT100;
   1:  PR[GP1:91,1] = PR[GP1:90,1] + -48.443;
   1:  PR[GP1:91,2] = PR[GP1:90,2] + 32.393;
   1:L PR[91] R[100]mm/sec CNT100;
   1:  PR[GP1:91,1] = PR[GP1:90,1] + -56.334;
   1:  PR[GP1:91,2] = PR[GP1:90,2] + 27.903;
   1:L PR[91] R[100]mm/sec CNT100;
   1:  PR[GP1:91,1] = PR[GP1:90,1] + -57.025;
   1:  PR[GP1:91,2] = PR[GP1:90,2] + 27.475;
   1:L PR[91] R[100]mm/sec CNT100;
   1:  PR[GP1:91,1] = PR[GP1:90,1] + -57.456;
   1:  PR[GP1:91,2] = PR[GP1:90,2] + 27.089;
   1:L PR[91] R[100]mm/sec CNT100;
   1:  PR[GP1:91,1] = PR[GP1:90,1] + -64.461;
   1:  PR[GP1:91,2] = PR[GP1:90,2] + 19.720;
   1:L PR[91] R[100]mm/sec CNT100;
   1:  PR[GP1:91,1] = PR[GP1:90,1] + -69.110;
   1:  PR[GP1:91,2] = PR[GP1:90,2] + 10.328;
   1:L PR[91] R[100]mm/sec CNT100;
   1:  PR[GP1:91,1] = PR[GP1:90,1] + -69.321;
   1:  PR[GP1:91,2] = PR[GP1:90,2] + 9.051;
   1:L PR[91] R[100]mm/sec CNT100;
   1:  PR[GP1:91,1] = PR[GP1:90,1] + -70.719;
   1:  PR[GP1:91,2] = PR[GP1:90,2] + -0.068;
   1:L PR[91] R[100]mm/sec CNT100;
   1:  PR[GP1:91,1] = PR[GP1:90,1] + -70.458;
   1:  PR[GP1:91,2] = PR[GP1:90,2] + -1.636;
   1:L PR[91] R[100]mm/sec CNT100;
   1:  PR[GP1:91,1] = PR[GP1:90,1] + -69.108;
   1:  PR[GP1:91,2] = PR[GP1:90,2] + -10.476;
   1:L PR[91] R[100]mm/sec CNT100;
   1:  PR[GP1:91,1] = PR[GP1:90,1] + -64.593;
   1:  PR[GP1:91,2] = PR[GP1:90,2] + -19.615;
   1:L PR[91] R[100]mm/sec CNT100;
   1:  PR[GP1:91,1] = PR[GP1:90,1] + -64.466;
   1:  PR[GP1:91,2] = PR[GP1:90,2] + -19.860;
   1:L PR[91] R[100]mm/sec CNT100;
   1:  PR[GP1:91,1] = PR[GP1:90,1] + -57.456;
   1:  PR[GP1:91,2] = PR[GP1:90,2] + -27.233;
   1:L PR[91] R[100]mm/sec CNT100;
   1:  PR[GP1:91,1] = PR[GP1:90,1] + -57.034;
   1:  PR[GP1:91,2] = PR[GP1:90,2] + -27.611;
   1:L PR[91] R[100]mm/sec CNT100;
   1:  PR[GP1:91,1] = PR[GP1:90,1] + -49.713;
   1:  PR[GP1:91,2] = PR[GP1:90,2] + -31.729;
   1:L PR[91] R[100]mm/sec CNT100;
   1:  PR[GP1:91,1] = PR[GP1:90,1] + -48.429;
   1:  PR[GP1:91,2] = PR[GP1:90,2] + -32.543;
   1:L PR[91] R[100]mm/sec CNT100;
   1:  PR[GP1:91,1] = PR[GP1:90,1] + -46.587;
   1:  PR[GP1:91,2] = PR[GP1:90,2] + -33.267;
   1:L PR[91] R[100]mm/sec CNT100;
   1:  PR[GP1:91,1] = PR[GP1:90,1] + -40.300;
   1:  PR[GP1:91,2] = PR[GP1:90,2] + -34.747;
   1:L PR[91] R[100]mm/sec CNT100;
   1:  PR[GP1:91,1] = PR[GP1:90,1] + -37.380;
   1:  PR[GP1:91,2] = PR[GP1:90,2] + -35.363;
   1:L PR[91] R[100]mm/sec CNT100;
   1:  PR[GP1:91,1] = PR[GP1:90,1] + -33.060;
   1:  PR[GP1:91,2] = PR[GP1:90,2] + -35.485;
   1:L PR[91] R[100]mm/sec CNT100;
   1:  PR[GP1:91,1] = PR[GP1:90,1] + -29.671;
   1:  PR[GP1:91,2] = PR[GP1:90,2] + -35.314;
   1:L PR[91] R[100]mm/sec CNT100;
   1:  PR[GP1:91,1] = PR[GP1:90,1] + -24.559;
   1:  PR[GP1:91,2] = PR[GP1:90,2] + -34.570;
   1:L PR[91] R[100]mm/sec CNT100;
   1:  PR[GP1:91,1] = PR[GP1:90,1] + -23.602;
   1:  PR[GP1:91,2] = PR[GP1:90,2] + -34.227;
   1:L PR[91] R[100]mm/sec CNT100;
   1:  PR[GP1:91,1] = PR[GP1:90,1] + -17.793;
   1:  PR[GP1:91,2] = PR[GP1:90,2] + -32.381;
   1:L PR[91] R[100]mm/sec CNT100;
   1:  PR[GP1:91,1] = PR[GP1:90,1] + -11.977;
   1:  PR[GP1:91,2] = PR[GP1:90,2] + -29.338;
   1:L PR[91] R[100]mm/sec CNT100;
   1:  PR[GP1:91,1] = PR[GP1:90,1] + -11.432;
   1:  PR[GP1:91,2] = PR[GP1:90,2] + -28.943;
   1:L PR[91] R[100]mm/sec CNT100;
   1:  PR[GP1:91,1] = PR[GP1:90,1] + -7.054;
   1:  PR[GP1:91,2] = PR[GP1:90,2] + -25.514;
   1:L PR[91] R[100]mm/sec CNT100;
   1:  PR[GP1:91,1] = PR[GP1:90,1] + -3.784;
   1:  PR[GP1:91,2] = PR[GP1:90,2] + -21.722;
   1:L PR[91] R[100]mm/sec CNT100;
   1:  PR[GP1:91,1] = PR[GP1:90,1] + -2.636;
   1:  PR[GP1:91,2] = PR[GP1:90,2] + -21.475;
   1:L PR[91] R[100]mm/sec CNT100;
   1:  PR[GP1:91,1] = PR[GP1:90,1] + 0.352;
   1:  PR[GP1:91,2] = PR[GP1:90,2] + -19.892;
   1:L PR[91] R[100]mm/sec CNT100;
   1:  PR[GP1:91,1] = PR[GP1:90,1] + 4.062;
   1:  PR[GP1:91,2] = PR[GP1:90,2] + -21.784;
   1:L PR[91] R[100]mm/sec CNT100;
   1:  PR[GP1:91,1] = PR[GP1:90,1] + 7.307;
   1:  PR[GP1:91,2] = PR[GP1:90,2] + -25.552;
   1:L PR[91] R[100]mm/sec CNT100;
   1:  PR[GP1:91,1] = PR[GP1:90,1] + 11.665;
   1:  PR[GP1:91,2] = PR[GP1:90,2] + -28.962;
   1:L PR[91] R[100]mm/sec CNT100;
   1:  PR[GP1:91,1] = PR[GP1:90,1] + 12.209;
   1:  PR[GP1:91,2] = PR[GP1:90,2] + -29.357;
   1:L PR[91] R[100]mm/sec CNT100;
   1:  PR[GP1:91,1] = PR[GP1:90,1] + 17.992;
   1:  PR[GP1:91,2] = PR[GP1:90,2] + -32.375;
   1:L PR[91] R[100]mm/sec CNT100;
   1:  PR[GP1:91,1] = PR[GP1:90,1] + 24.759;
   1:  PR[GP1:91,2] = PR[GP1:90,2] + -34.565;
   1:L PR[91] R[100]mm/sec CNT100;
   1:  PR[GP1:91,1] = PR[GP1:90,1] + 29.876;
   1:  PR[GP1:91,2] = PR[GP1:90,2] + -35.313;
   1:L PR[91] R[100]mm/sec CNT100;
   1:  PR[GP1:91,1] = PR[GP1:90,1] + 33.262;
   1:  PR[GP1:91,2] = PR[GP1:90,2] + -35.486;
   1:L PR[91] R[100]mm/sec CNT100;
   1:  PR[GP1:91,1] = PR[GP1:90,1] + 37.565;
   1:  PR[GP1:91,2] = PR[GP1:90,2] + -35.366;
   1:L PR[91] R[100]mm/sec CNT100;
   1:  PR[GP1:91,1] = PR[GP1:90,1] + 43.869;
   1:  PR[GP1:91,2] = PR[GP1:90,2] + -33.899;
   1:L PR[91] R[100]mm/sec CNT100;
   1:  PR[GP1:91,1] = PR[GP1:90,1] + 46.789;
   1:  PR[GP1:91,2] = PR[GP1:90,2] + -33.267;
   1:L PR[91] R[100]mm/sec CNT100;
   1:  PR[GP1:91,1] = PR[GP1:90,1] + 48.647;
   1:  PR[GP1:91,2] = PR[GP1:90,2] + -32.540;
   1:L PR[91] R[100]mm/sec CNT100;
   1:  PR[GP1:91,1] = PR[GP1:90,1] + 56.542;
   1:  PR[GP1:91,2] = PR[GP1:90,2] + -28.055;
   1:L PR[91] R[100]mm/sec CNT100;
   1:  PR[GP1:91,1] = PR[GP1:90,1] + 57.231;
   1:  PR[GP1:91,2] = PR[GP1:90,2] + -27.630;
   1:L PR[91] R[100]mm/sec CNT100;
   1:  PR[GP1:91,1] = PR[GP1:90,1] + 57.661;
   1:  PR[GP1:91,2] = PR[GP1:90,2] + -27.246;
   1:L PR[91] R[100]mm/sec CNT100;
   1:  PR[GP1:91,1] = PR[GP1:90,1] + 64.674;
   1:  PR[GP1:91,2] = PR[GP1:90,2] + -19.847;
   1:L PR[91] R[100]mm/sec CNT100;
   1:  PR[GP1:91,1] = PR[GP1:90,1] + 69.323;
   1:  PR[GP1:91,2] = PR[GP1:90,2] + -10.500;
   1:L PR[91] R[100]mm/sec CNT100;
   1:  PR[GP1:91,1] = PR[GP1:90,1] + 69.534;
   1:  PR[GP1:91,2] = PR[GP1:90,2] + -9.222;
   1:L PR[91] R[100]mm/sec CNT100;
   1:  PR[GP1:91,1] = PR[GP1:90,1] + 70.932;
   1:  PR[GP1:91,2] = PR[GP1:90,2] + -0.076;
   1:L PR[91] R[100]mm/sec CNT100;
   1:  PR[GP1:91,1] = PR[GP1:90,1] + 70.671;
   1:  PR[GP1:91,2] = PR[GP1:90,2] + 1.495;
   1:L PR[91] R[100]mm/sec CNT100;
   1:  PR[GP1:91,1] = PR[GP1:90,1] + 69.321;
   1:  PR[GP1:91,2] = PR[GP1:90,2] + 10.359;
   1:L PR[91] R[100]mm/sec CNT100;
   1:  PR[GP1:91,1] = PR[GP1:90,1] + 64.674;
   1:  PR[GP1:91,2] = PR[GP1:90,2] + 19.703;
   1:L PR[91] R[100]mm/sec CNT100;
   1:  PR[GP1:91,1] = PR[GP1:90,1] + 57.661;
   1:  PR[GP1:91,2] = PR[GP1:90,2] + 27.102;
   1:L PR[91] R[100]mm/sec CNT100;
   1:  PR[GP1:91,1] = PR[GP1:90,1] + 57.241;
   1:  PR[GP1:91,2] = PR[GP1:90,2] + 27.478;
   1:L PR[91] R[100]mm/sec CNT100;
   1:  PR[GP1:91,1] = PR[GP1:90,1] + 49.914;
   1:  PR[GP1:91,2] = PR[GP1:90,2] + 31.594;
   1:L PR[91] R[100]mm/sec CNT100;
   1:  PR[GP1:91,1] = PR[GP1:90,1] + 48.634;
   1:  PR[GP1:91,2] = PR[GP1:90,2] + 32.401;
   1:L PR[91] R[100]mm/sec CNT100;
   1:  PR[GP1:91,1] = PR[GP1:90,1] + 46.784;
   1:  PR[GP1:91,2] = PR[GP1:90,2] + 33.125;
   1:L PR[91] R[100]mm/sec CNT100;
   1:  PR[GP1:91,1] = PR[GP1:90,1] + 40.495;
   1:  PR[GP1:91,2] = PR[GP1:90,2] + 34.608;
   1:L PR[91] R[100]mm/sec CNT100;
   1:  PR[GP1:91,1] = PR[GP1:90,1] + 37.571;
   1:  PR[GP1:91,2] = PR[GP1:90,2] + 35.222;
   1:L PR[91] R[100]mm/sec CNT100;
   1:  PR[GP1:91,1] = PR[GP1:90,1] + 33.262;
   1:  PR[GP1:91,2] = PR[GP1:90,2] + 35.342;
   1:L PR[91] R[100]mm/sec CNT100;
   1:  PR[GP1:91,1] = PR[GP1:90,1] + 29.876;
   1:  PR[GP1:91,2] = PR[GP1:90,2] + 35.169;
   1:L PR[91] R[100]mm/sec CNT100;
   1:  PR[GP1:91,1] = PR[GP1:90,1] + 24.768;
   1:  PR[GP1:91,2] = PR[GP1:90,2] + 34.422;
   1:L PR[91] R[100]mm/sec CNT100;
   1:  PR[GP1:91,1] = PR[GP1:90,1] + 23.811;
   1:  PR[GP1:91,2] = PR[GP1:90,2] + 34.080;
   1:L PR[91] R[100]mm/sec CNT100;
   1:  PR[GP1:91,1] = PR[GP1:90,1] + 17.991;
   1:  PR[GP1:91,2] = PR[GP1:90,2] + 32.230;
   1:L PR[91] R[100]mm/sec CNT100;
   1:  PR[GP1:91,1] = PR[GP1:90,1] + 12.207;
   1:  PR[GP1:91,2] = PR[GP1:90,2] + 29.212;
   1:L PR[91] R[100]mm/sec CNT100;
   1:  PR[GP1:91,1] = PR[GP1:90,1] + 11.823;
   1:  PR[GP1:91,2] = PR[GP1:90,2] + 28.941;
   1:L PR[91] R[100]mm/sec CNT100;
   1:  PR[GP1:91,1] = PR[GP1:90,1] + 7.408;
   1:  PR[GP1:91,2] = PR[GP1:90,2] + 25.486;
   1:L PR[91] R[100]mm/sec CNT100;
   1:  PR[GP1:91,1] = PR[GP1:90,1] + 4.043;
   1:  PR[GP1:91,2] = PR[GP1:90,2] + 21.570;
   1:L PR[91] R[100]mm/sec CNT100;
   1:  PR[GP1:91,1] = PR[GP1:90,1] + 3.490;
   1:  PR[GP1:91,2] = PR[GP1:90,2] + 21.352;
   1:L PR[91] R[100]mm/sec CNT100;
   1:  PR[GP1:91,1] = PR[GP1:90,1] + 0.465;
   1:  PR[GP1:91,2] = PR[GP1:90,2] + 19.805;
   1:L PR[91] R[100]mm/sec CNT100;
   1:  ! -- Layer/Ebene 69 -- !;
   1:  PR[91] = PR[90];
   1:  PR[GP1:91,1] = PR[GP1:90,1] + -0.679;
   1:  PR[GP1:91,2] = PR[GP1:90,2] + 20.288;
   1:  PR[GP1:91,3] = PR[GP1:90,3] + 42.395;
   1:L PR[91] R[100]mm/sec CNT100;
   1:  PR[GP1:91,1] = PR[GP1:90,1] + -3.811;
   1:  PR[GP1:91,2] = PR[GP1:90,2] + 21.880;
   1:L PR[91] R[100]mm/sec CNT100;
   1:  PR[GP1:91,1] = PR[GP1:90,1] + -6.998;
   1:  PR[GP1:91,2] = PR[GP1:90,2] + 25.587;
   1:L PR[91] R[100]mm/sec CNT100;
   1:  PR[GP1:91,1] = PR[GP1:90,1] + -11.261;
   1:  PR[GP1:91,2] = PR[GP1:90,2] + 28.925;
   1:L PR[91] R[100]mm/sec CNT100;
   1:  PR[GP1:91,1] = PR[GP1:90,1] + -11.763;
   1:  PR[GP1:91,2] = PR[GP1:90,2] + 29.280;
   1:L PR[91] R[100]mm/sec CNT100;
   1:  PR[GP1:91,1] = PR[GP1:90,1] + -17.453;
   1:  PR[GP1:91,2] = PR[GP1:90,2] + 32.257;
   1:L PR[91] R[100]mm/sec CNT100;
   1:  PR[GP1:91,1] = PR[GP1:90,1] + -24.248;
   1:  PR[GP1:91,2] = PR[GP1:90,2] + 34.446;
   1:L PR[91] R[100]mm/sec CNT100;
   1:  PR[GP1:91,1] = PR[GP1:90,1] + -29.811;
   1:  PR[GP1:91,2] = PR[GP1:90,2] + 35.255;
   1:L PR[91] R[100]mm/sec CNT100;
   1:  PR[GP1:91,1] = PR[GP1:90,1] + -32.409;
   1:  PR[GP1:91,2] = PR[GP1:90,2] + 35.387;
   1:L PR[91] R[100]mm/sec CNT100;
   1:  PR[GP1:91,1] = PR[GP1:90,1] + -37.254;
   1:  PR[GP1:91,2] = PR[GP1:90,2] + 35.249;
   1:L PR[91] R[100]mm/sec CNT100;
   1:  PR[GP1:91,1] = PR[GP1:90,1] + -42.676;
   1:  PR[GP1:91,2] = PR[GP1:90,2] + 33.988;
   1:L PR[91] R[100]mm/sec CNT100;
   1:  PR[GP1:91,1] = PR[GP1:90,1] + -46.198;
   1:  PR[GP1:91,2] = PR[GP1:90,2] + 33.225;
   1:L PR[91] R[100]mm/sec CNT100;
   1:  PR[GP1:91,1] = PR[GP1:90,1] + -48.447;
   1:  PR[GP1:91,2] = PR[GP1:90,2] + 32.340;
   1:L PR[91] R[100]mm/sec CNT100;
   1:  PR[GP1:91,1] = PR[GP1:90,1] + -55.710;
   1:  PR[GP1:91,2] = PR[GP1:90,2] + 28.207;
   1:L PR[91] R[100]mm/sec CNT100;
   1:  PR[GP1:91,1] = PR[GP1:90,1] + -56.812;
   1:  PR[GP1:91,2] = PR[GP1:90,2] + 27.525;
   1:L PR[91] R[100]mm/sec CNT100;
   1:  PR[GP1:91,1] = PR[GP1:90,1] + -57.512;
   1:  PR[GP1:91,2] = PR[GP1:90,2] + 26.898;
   1:L PR[91] R[100]mm/sec CNT100;
   1:  PR[GP1:91,1] = PR[GP1:90,1] + -64.297;
   1:  PR[GP1:91,2] = PR[GP1:90,2] + 19.764;
   1:L PR[91] R[100]mm/sec CNT100;
   1:  PR[GP1:91,1] = PR[GP1:90,1] + -64.346;
   1:  PR[GP1:91,2] = PR[GP1:90,2] + 19.700;
   1:L PR[91] R[100]mm/sec CNT100;
   1:  PR[GP1:91,1] = PR[GP1:90,1] + -65.652;
   1:  PR[GP1:91,2] = PR[GP1:90,2] + 17.088;
   1:L PR[91] R[100]mm/sec CNT100;
   1:  PR[GP1:91,1] = PR[GP1:90,1] + -69.000;
   1:  PR[GP1:91,2] = PR[GP1:90,2] + 10.310;
   1:L PR[91] R[100]mm/sec CNT100;
   1:  PR[GP1:91,1] = PR[GP1:90,1] + -70.600;
   1:  PR[GP1:91,2] = PR[GP1:90,2] + -0.068;
   1:L PR[91] R[100]mm/sec CNT100;
   1:  PR[GP1:91,1] = PR[GP1:90,1] + -70.431;
   1:  PR[GP1:91,2] = PR[GP1:90,2] + -1.082;
   1:L PR[91] R[100]mm/sec CNT100;
   1:  PR[GP1:91,1] = PR[GP1:90,1] + -69.000;
   1:  PR[GP1:91,2] = PR[GP1:90,2] + -10.455;
   1:L PR[91] R[100]mm/sec CNT100;
   1:  PR[GP1:91,1] = PR[GP1:90,1] + -65.652;
   1:  PR[GP1:91,2] = PR[GP1:90,2] + -17.232;
   1:L PR[91] R[100]mm/sec CNT100;
   1:  PR[GP1:91,1] = PR[GP1:90,1] + -64.346;
   1:  PR[GP1:91,2] = PR[GP1:90,2] + -19.844;
   1:L PR[91] R[100]mm/sec CNT100;
   1:  PR[GP1:91,1] = PR[GP1:90,1] + -64.297;
   1:  PR[GP1:91,2] = PR[GP1:90,2] + -19.908;
   1:L PR[91] R[100]mm/sec CNT100;
   1:  PR[GP1:91,1] = PR[GP1:90,1] + -57.512;
   1:  PR[GP1:91,2] = PR[GP1:90,2] + -27.042;
   1:L PR[91] R[100]mm/sec CNT100;
   1:  PR[GP1:91,1] = PR[GP1:90,1] + -56.821;
   1:  PR[GP1:91,2] = PR[GP1:90,2] + -27.660;
   1:L PR[91] R[100]mm/sec CNT100;
   1:  PR[GP1:91,1] = PR[GP1:90,1] + -49.989;
   1:  PR[GP1:91,2] = PR[GP1:90,2] + -31.504;
   1:L PR[91] R[100]mm/sec CNT100;
   1:  PR[GP1:91,1] = PR[GP1:90,1] + -48.433;
   1:  PR[GP1:91,2] = PR[GP1:90,2] + -32.489;
   1:L PR[91] R[100]mm/sec CNT100;
   1:  PR[GP1:91,1] = PR[GP1:90,1] + -46.193;
   1:  PR[GP1:91,2] = PR[GP1:90,2] + -33.371;
   1:L PR[91] R[100]mm/sec CNT100;
   1:  PR[GP1:91,1] = PR[GP1:90,1] + -40.540;
   1:  PR[GP1:91,2] = PR[GP1:90,2] + -34.702;
   1:L PR[91] R[100]mm/sec CNT100;
   1:  PR[GP1:91,1] = PR[GP1:90,1] + -37.261;
   1:  PR[GP1:91,2] = PR[GP1:90,2] + -35.393;
   1:L PR[91] R[100]mm/sec CNT100;
   1:  PR[GP1:91,1] = PR[GP1:90,1] + -32.409;
   1:  PR[GP1:91,2] = PR[GP1:90,2] + -35.531;
   1:L PR[91] R[100]mm/sec CNT100;
   1:  PR[GP1:91,1] = PR[GP1:90,1] + -29.811;
   1:  PR[GP1:91,2] = PR[GP1:90,2] + -35.399;
   1:L PR[91] R[100]mm/sec CNT100;
   1:  PR[GP1:91,1] = PR[GP1:90,1] + -24.258;
   1:  PR[GP1:91,2] = PR[GP1:90,2] + -34.591;
   1:L PR[91] R[100]mm/sec CNT100;
   1:  PR[GP1:91,1] = PR[GP1:90,1] + -23.949;
   1:  PR[GP1:91,2] = PR[GP1:90,2] + -34.481;
   1:L PR[91] R[100]mm/sec CNT100;
   1:  PR[GP1:91,1] = PR[GP1:90,1] + -17.993;
   1:  PR[GP1:91,2] = PR[GP1:90,2] + -32.589;
   1:L PR[91] R[100]mm/sec CNT100;
   1:  PR[GP1:91,1] = PR[GP1:90,1] + -17.458;
   1:  PR[GP1:91,2] = PR[GP1:90,2] + -32.403;
   1:L PR[91] R[100]mm/sec CNT100;
   1:  PR[GP1:91,1] = PR[GP1:90,1] + -11.766;
   1:  PR[GP1:91,2] = PR[GP1:90,2] + -29.425;
   1:L PR[91] R[100]mm/sec CNT100;
   1:  PR[GP1:91,1] = PR[GP1:90,1] + -11.058;
   1:  PR[GP1:91,2] = PR[GP1:90,2] + -28.911;
   1:L PR[91] R[100]mm/sec CNT100;
   1:  PR[GP1:91,1] = PR[GP1:90,1] + -6.881;
   1:  PR[GP1:91,2] = PR[GP1:90,2] + -25.640;
   1:L PR[91] R[100]mm/sec CNT100;
   1:  PR[GP1:91,1] = PR[GP1:90,1] + -3.755;
   1:  PR[GP1:91,2] = PR[GP1:90,2] + -22.015;
   1:L PR[91] R[100]mm/sec CNT100;
   1:  PR[GP1:91,1] = PR[GP1:90,1] + -2.469;
   1:  PR[GP1:91,2] = PR[GP1:90,2] + -21.738;
   1:L PR[91] R[100]mm/sec CNT100;
   1:  PR[GP1:91,1] = PR[GP1:90,1] + 0.393;
   1:  PR[GP1:91,2] = PR[GP1:90,2] + -20.222;
   1:L PR[91] R[100]mm/sec CNT100;
   1:  PR[GP1:91,1] = PR[GP1:90,1] + 4.032;
   1:  PR[GP1:91,2] = PR[GP1:90,2] + -22.077;
   1:L PR[91] R[100]mm/sec CNT100;
   1:  PR[GP1:91,1] = PR[GP1:90,1] + 7.131;
   1:  PR[GP1:91,2] = PR[GP1:90,2] + -25.676;
   1:L PR[91] R[100]mm/sec CNT100;
   1:  PR[GP1:91,1] = PR[GP1:90,1] + 11.290;
   1:  PR[GP1:91,2] = PR[GP1:90,2] + -28.930;
   1:L PR[91] R[100]mm/sec CNT100;
   1:  PR[GP1:91,1] = PR[GP1:90,1] + 11.998;
   1:  PR[GP1:91,2] = PR[GP1:90,2] + -29.444;
   1:L PR[91] R[100]mm/sec CNT100;
   1:  PR[GP1:91,1] = PR[GP1:90,1] + 17.649;
   1:  PR[GP1:91,2] = PR[GP1:90,2] + -32.393;
   1:L PR[91] R[100]mm/sec CNT100;
   1:  PR[GP1:91,1] = PR[GP1:90,1] + 24.456;
   1:  PR[GP1:91,2] = PR[GP1:90,2] + -34.586;
   1:L PR[91] R[100]mm/sec CNT100;
   1:  PR[GP1:91,1] = PR[GP1:90,1] + 30.015;
   1:  PR[GP1:91,2] = PR[GP1:90,2] + -35.399;
   1:L PR[91] R[100]mm/sec CNT100;
   1:  PR[GP1:91,1] = PR[GP1:90,1] + 32.610;
   1:  PR[GP1:91,2] = PR[GP1:90,2] + -35.531;
   1:L PR[91] R[100]mm/sec CNT100;
   1:  PR[GP1:91,1] = PR[GP1:90,1] + 37.442;
   1:  PR[GP1:91,2] = PR[GP1:90,2] + -35.397;
   1:L PR[91] R[100]mm/sec CNT100;
   1:  PR[GP1:91,1] = PR[GP1:90,1] + 42.861;
   1:  PR[GP1:91,2] = PR[GP1:90,2] + -34.136;
   1:L PR[91] R[100]mm/sec CNT100;
   1:  PR[GP1:91,1] = PR[GP1:90,1] + 46.391;
   1:  PR[GP1:91,2] = PR[GP1:90,2] + -33.372;
   1:L PR[91] R[100]mm/sec CNT100;
   1:  PR[GP1:91,1] = PR[GP1:90,1] + 48.650;
   1:  PR[GP1:91,2] = PR[GP1:90,2] + -32.488;
   1:L PR[91] R[100]mm/sec CNT100;
   1:  PR[GP1:91,1] = PR[GP1:90,1] + 55.915;
   1:  PR[GP1:91,2] = PR[GP1:90,2] + -28.360;
   1:L PR[91] R[100]mm/sec CNT100;
   1:  PR[GP1:91,1] = PR[GP1:90,1] + 57.014;
   1:  PR[GP1:91,2] = PR[GP1:90,2] + -27.683;
   1:L PR[91] R[100]mm/sec CNT100;
   1:  PR[GP1:91,1] = PR[GP1:90,1] + 57.713;
   1:  PR[GP1:91,2] = PR[GP1:90,2] + -27.058;
   1:L PR[91] R[100]mm/sec CNT100;
   1:  PR[GP1:91,1] = PR[GP1:90,1] + 64.507;
   1:  PR[GP1:91,2] = PR[GP1:90,2] + -19.894;
   1:L PR[91] R[100]mm/sec CNT100;
   1:  PR[GP1:91,1] = PR[GP1:90,1] + 64.558;
   1:  PR[GP1:91,2] = PR[GP1:90,2] + -19.827;
   1:L PR[91] R[100]mm/sec CNT100;
   1:  PR[GP1:91,1] = PR[GP1:90,1] + 65.866;
   1:  PR[GP1:91,2] = PR[GP1:90,2] + -17.224;
   1:L PR[91] R[100]mm/sec CNT100;
   1:  PR[GP1:91,1] = PR[GP1:90,1] + 69.213;
   1:  PR[GP1:91,2] = PR[GP1:90,2] + -10.483;
   1:L PR[91] R[100]mm/sec CNT100;
   1:  PR[GP1:91,1] = PR[GP1:90,1] + 70.813;
   1:  PR[GP1:91,2] = PR[GP1:90,2] + -0.076;
   1:L PR[91] R[100]mm/sec CNT100;
   1:  PR[GP1:91,1] = PR[GP1:90,1] + 70.644;
   1:  PR[GP1:91,2] = PR[GP1:90,2] + 0.940;
   1:L PR[91] R[100]mm/sec CNT100;
   1:  PR[GP1:91,1] = PR[GP1:90,1] + 69.213;
   1:  PR[GP1:91,2] = PR[GP1:90,2] + 10.339;
   1:L PR[91] R[100]mm/sec CNT100;
   1:  PR[GP1:91,1] = PR[GP1:90,1] + 65.866;
   1:  PR[GP1:91,2] = PR[GP1:90,2] + 17.080;
   1:L PR[91] R[100]mm/sec CNT100;
   1:  PR[GP1:91,1] = PR[GP1:90,1] + 64.558;
   1:  PR[GP1:91,2] = PR[GP1:90,2] + 19.683;
   1:L PR[91] R[100]mm/sec CNT100;
   1:  PR[GP1:91,1] = PR[GP1:90,1] + 64.507;
   1:  PR[GP1:91,2] = PR[GP1:90,2] + 19.750;
   1:L PR[91] R[100]mm/sec CNT100;
   1:  PR[GP1:91,1] = PR[GP1:90,1] + 57.713;
   1:  PR[GP1:91,2] = PR[GP1:90,2] + 26.914;
   1:L PR[91] R[100]mm/sec CNT100;
   1:  PR[GP1:91,1] = PR[GP1:90,1] + 57.023;
   1:  PR[GP1:91,2] = PR[GP1:90,2] + 27.531;
   1:L PR[91] R[100]mm/sec CNT100;
   1:  PR[GP1:91,1] = PR[GP1:90,1] + 50.187;
   1:  PR[GP1:91,2] = PR[GP1:90,2] + 31.372;
   1:L PR[91] R[100]mm/sec CNT100;
   1:  PR[GP1:91,1] = PR[GP1:90,1] + 48.637;
   1:  PR[GP1:91,2] = PR[GP1:90,2] + 32.349;
   1:L PR[91] R[100]mm/sec CNT100;
   1:  PR[GP1:91,1] = PR[GP1:90,1] + 46.386;
   1:  PR[GP1:91,2] = PR[GP1:90,2] + 33.230;
   1:L PR[91] R[100]mm/sec CNT100;
   1:  PR[GP1:91,1] = PR[GP1:90,1] + 40.733;
   1:  PR[GP1:91,2] = PR[GP1:90,2] + 34.562;
   1:L PR[91] R[100]mm/sec CNT100;
   1:  PR[GP1:91,1] = PR[GP1:90,1] + 37.449;
   1:  PR[GP1:91,2] = PR[GP1:90,2] + 35.253;
   1:L PR[91] R[100]mm/sec CNT100;
   1:  PR[GP1:91,1] = PR[GP1:90,1] + 32.610;
   1:  PR[GP1:91,2] = PR[GP1:90,2] + 35.387;
   1:L PR[91] R[100]mm/sec CNT100;
   1:  PR[GP1:91,1] = PR[GP1:90,1] + 30.015;
   1:  PR[GP1:91,2] = PR[GP1:90,2] + 35.255;
   1:L PR[91] R[100]mm/sec CNT100;
   1:  PR[GP1:91,1] = PR[GP1:90,1] + 24.466;
   1:  PR[GP1:91,2] = PR[GP1:90,2] + 34.443;
   1:L PR[91] R[100]mm/sec CNT100;
   1:  PR[GP1:91,1] = PR[GP1:90,1] + 24.158;
   1:  PR[GP1:91,2] = PR[GP1:90,2] + 34.333;
   1:L PR[91] R[100]mm/sec CNT100;
   1:  PR[GP1:91,1] = PR[GP1:90,1] + 18.193;
   1:  PR[GP1:91,2] = PR[GP1:90,2] + 32.439;
   1:L PR[91] R[100]mm/sec CNT100;
   1:  PR[GP1:91,1] = PR[GP1:90,1] + 17.656;
   1:  PR[GP1:91,2] = PR[GP1:90,2] + 32.253;
   1:L PR[91] R[100]mm/sec CNT100;
   1:  PR[GP1:91,1] = PR[GP1:90,1] + 11.995;
   1:  PR[GP1:91,2] = PR[GP1:90,2] + 29.299;
   1:L PR[91] R[100]mm/sec CNT100;
   1:  PR[GP1:91,1] = PR[GP1:90,1] + 11.492;
   1:  PR[GP1:91,2] = PR[GP1:90,2] + 28.943;
   1:L PR[91] R[100]mm/sec CNT100;
   1:  PR[GP1:91,1] = PR[GP1:90,1] + 7.250;
   1:  PR[GP1:91,2] = PR[GP1:90,2] + 25.624;
   1:L PR[91] R[100]mm/sec CNT100;
   1:  PR[GP1:91,1] = PR[GP1:90,1] + 4.014;
   1:  PR[GP1:91,2] = PR[GP1:90,2] + 21.857;
   1:L PR[91] R[100]mm/sec CNT100;
   1:  PR[GP1:91,1] = PR[GP1:90,1] + 3.401;
   1:  PR[GP1:91,2] = PR[GP1:90,2] + 21.615;
   1:L PR[91] R[100]mm/sec CNT100;
   1:  PR[GP1:91,1] = PR[GP1:90,1] + 0.506;
   1:  PR[GP1:91,2] = PR[GP1:90,2] + 20.135;
   1:L PR[91] R[100]mm/sec CNT100;
   1:  ! -- Layer/Ebene 70 -- !;
   1:  PR[91] = PR[90];
   1:  PR[GP1:91,1] = PR[GP1:90,1] + -0.768;
   1:  PR[GP1:91,2] = PR[GP1:90,2] + 20.634;
   1:  PR[GP1:91,3] = PR[GP1:90,3] + 43.005;
   1:L PR[91] R[100]mm/sec CNT100;
   1:  PR[GP1:91,1] = PR[GP1:90,1] + -3.781;
   1:  PR[GP1:91,2] = PR[GP1:90,2] + 22.167;
   1:L PR[91] R[100]mm/sec CNT100;
   1:  PR[GP1:91,1] = PR[GP1:90,1] + -6.843;
   1:  PR[GP1:91,2] = PR[GP1:90,2] + 25.726;
   1:L PR[91] R[100]mm/sec CNT100;
   1:  PR[GP1:91,1] = PR[GP1:90,1] + -10.931;
   1:  PR[GP1:91,2] = PR[GP1:90,2] + 28.928;
   1:L PR[91] R[100]mm/sec CNT100;
   1:  PR[GP1:91,1] = PR[GP1:90,1] + -11.553;
   1:  PR[GP1:91,2] = PR[GP1:90,2] + 29.368;
   1:L PR[91] R[100]mm/sec CNT100;
   1:  PR[GP1:91,1] = PR[GP1:90,1] + -17.111;
   1:  PR[GP1:91,2] = PR[GP1:90,2] + 32.275;
   1:L PR[91] R[100]mm/sec CNT100;
   1:  PR[GP1:91,1] = PR[GP1:90,1] + -23.989;
   1:  PR[GP1:91,2] = PR[GP1:90,2] + 34.489;
   1:L PR[91] R[100]mm/sec CNT100;
   1:  PR[GP1:91,1] = PR[GP1:90,1] + -25.043;
   1:  PR[GP1:91,2] = PR[GP1:90,2] + 34.626;
   1:L PR[91] R[100]mm/sec CNT100;
   1:  PR[GP1:91,1] = PR[GP1:90,1] + -29.951;
   1:  PR[GP1:91,2] = PR[GP1:90,2] + 35.340;
   1:L PR[91] R[100]mm/sec CNT100;
   1:  PR[GP1:91,1] = PR[GP1:90,1] + -31.758;
   1:  PR[GP1:91,2] = PR[GP1:90,2] + 35.432;
   1:L PR[91] R[100]mm/sec CNT100;
   1:  PR[GP1:91,1] = PR[GP1:90,1] + -37.135;
   1:  PR[GP1:91,2] = PR[GP1:90,2] + 35.279;
   1:L PR[91] R[100]mm/sec CNT100;
   1:  PR[GP1:91,1] = PR[GP1:90,1] + -41.673;
   1:  PR[GP1:91,2] = PR[GP1:90,2] + 34.224;
   1:L PR[91] R[100]mm/sec CNT100;
   1:  PR[GP1:91,1] = PR[GP1:90,1] + -45.804;
   1:  PR[GP1:91,2] = PR[GP1:90,2] + 33.329;
   1:L PR[91] R[100]mm/sec CNT100;
   1:  PR[GP1:91,1] = PR[GP1:90,1] + -48.451;
   1:  PR[GP1:91,2] = PR[GP1:90,2] + 32.287;
   1:L PR[91] R[100]mm/sec CNT100;
   1:  PR[GP1:91,1] = PR[GP1:90,1] + -55.086;
   1:  PR[GP1:91,2] = PR[GP1:90,2] + 28.512;
   1:L PR[91] R[100]mm/sec CNT100;
   1:  PR[GP1:91,1] = PR[GP1:90,1] + -56.598;
   1:  PR[GP1:91,2] = PR[GP1:90,2] + 27.575;
   1:L PR[91] R[100]mm/sec CNT100;
   1:  PR[GP1:91,1] = PR[GP1:90,1] + -57.567;
   1:  PR[GP1:91,2] = PR[GP1:90,2] + 26.706;
   1:L PR[91] R[100]mm/sec CNT100;
   1:  PR[GP1:91,1] = PR[GP1:90,1] + -63.930;
   1:  PR[GP1:91,2] = PR[GP1:90,2] + 20.017;
   1:L PR[91] R[100]mm/sec CNT100;
   1:  PR[GP1:91,1] = PR[GP1:90,1] + -64.221;
   1:  PR[GP1:91,2] = PR[GP1:90,2] + 19.639;
   1:L PR[91] R[100]mm/sec CNT100;
   1:  PR[GP1:91,1] = PR[GP1:90,1] + -68.892;
   1:  PR[GP1:91,2] = PR[GP1:90,2] + 10.288;
   1:L PR[91] R[100]mm/sec CNT100;
   1:  PR[GP1:91,1] = PR[GP1:90,1] + -70.480;
   1:  PR[GP1:91,2] = PR[GP1:90,2] + -0.068;
   1:L PR[91] R[100]mm/sec CNT100;
   1:  PR[GP1:91,1] = PR[GP1:90,1] + -70.404;
   1:  PR[GP1:91,2] = PR[GP1:90,2] + -0.527;
   1:L PR[91] R[100]mm/sec CNT100;
   1:  PR[GP1:91,1] = PR[GP1:90,1] + -68.892;
   1:  PR[GP1:91,2] = PR[GP1:90,2] + -10.433;
   1:L PR[91] R[100]mm/sec CNT100;
   1:  PR[GP1:91,1] = PR[GP1:90,1] + -64.221;
   1:  PR[GP1:91,2] = PR[GP1:90,2] + -19.783;
   1:L PR[91] R[100]mm/sec CNT100;
   1:  PR[GP1:91,1] = PR[GP1:90,1] + -63.930;
   1:  PR[GP1:91,2] = PR[GP1:90,2] + -20.161;
   1:L PR[91] R[100]mm/sec CNT100;
   1:  PR[GP1:91,1] = PR[GP1:90,1] + -57.567;
   1:  PR[GP1:91,2] = PR[GP1:90,2] + -26.850;
   1:L PR[91] R[100]mm/sec CNT100;
   1:  PR[GP1:91,1] = PR[GP1:90,1] + -56.608;
   1:  PR[GP1:91,2] = PR[GP1:90,2] + -27.710;
   1:L PR[91] R[100]mm/sec CNT100;
   1:  PR[GP1:91,1] = PR[GP1:90,1] + -50.265;
   1:  PR[GP1:91,2] = PR[GP1:90,2] + -31.279;
   1:L PR[91] R[100]mm/sec CNT100;
   1:  PR[GP1:91,1] = PR[GP1:90,1] + -48.438;
   1:  PR[GP1:91,2] = PR[GP1:90,2] + -32.436;
   1:L PR[91] R[100]mm/sec CNT100;
   1:  PR[GP1:91,1] = PR[GP1:90,1] + -45.799;
   1:  PR[GP1:91,2] = PR[GP1:90,2] + -33.475;
   1:L PR[91] R[100]mm/sec CNT100;
   1:  PR[GP1:91,1] = PR[GP1:90,1] + -40.780;
   1:  PR[GP1:91,2] = PR[GP1:90,2] + -34.656;
   1:L PR[91] R[100]mm/sec CNT100;
   1:  PR[GP1:91,1] = PR[GP1:90,1] + -37.141;
   1:  PR[GP1:91,2] = PR[GP1:90,2] + -35.423;
   1:L PR[91] R[100]mm/sec CNT100;
   1:  PR[GP1:91,1] = PR[GP1:90,1] + -31.758;
   1:  PR[GP1:91,2] = PR[GP1:90,2] + -35.576;
   1:L PR[91] R[100]mm/sec CNT100;
   1:  PR[GP1:91,1] = PR[GP1:90,1] + -29.951;
   1:  PR[GP1:91,2] = PR[GP1:90,2] + -35.484;
   1:L PR[91] R[100]mm/sec CNT100;
   1:  PR[GP1:91,1] = PR[GP1:90,1] + -25.043;
   1:  PR[GP1:91,2] = PR[GP1:90,2] + -34.770;
   1:L PR[91] R[100]mm/sec CNT100;
   1:  PR[GP1:91,1] = PR[GP1:90,1] + -23.988;
   1:  PR[GP1:91,2] = PR[GP1:90,2] + -34.633;
   1:L PR[91] R[100]mm/sec CNT100;
   1:  PR[GP1:91,1] = PR[GP1:90,1] + -17.924;
   1:  PR[GP1:91,2] = PR[GP1:90,2] + -32.703;
   1:L PR[91] R[100]mm/sec CNT100;
   1:  PR[GP1:91,1] = PR[GP1:90,1] + -17.116;
   1:  PR[GP1:91,2] = PR[GP1:90,2] + -32.422;
   1:L PR[91] R[100]mm/sec CNT100;
   1:  PR[GP1:91,1] = PR[GP1:90,1] + -11.555;
   1:  PR[GP1:91,2] = PR[GP1:90,2] + -29.512;
   1:L PR[91] R[100]mm/sec CNT100;
   1:  PR[GP1:91,1] = PR[GP1:90,1] + -10.684;
   1:  PR[GP1:91,2] = PR[GP1:90,2] + -28.880;
   1:L PR[91] R[100]mm/sec CNT100;
   1:  PR[GP1:91,1] = PR[GP1:90,1] + -6.707;
   1:  PR[GP1:91,2] = PR[GP1:90,2] + -25.766;
   1:L PR[91] R[100]mm/sec CNT100;
   1:  PR[GP1:91,1] = PR[GP1:90,1] + -3.726;
   1:  PR[GP1:91,2] = PR[GP1:90,2] + -22.308;
   1:L PR[91] R[100]mm/sec CNT100;
   1:  PR[GP1:91,1] = PR[GP1:90,1] + -2.302;
   1:  PR[GP1:91,2] = PR[GP1:90,2] + -22.002;
   1:L PR[91] R[100]mm/sec CNT100;
   1:  PR[GP1:91,1] = PR[GP1:90,1] + 0.434;
   1:  PR[GP1:91,2] = PR[GP1:90,2] + -20.552;
   1:L PR[91] R[100]mm/sec CNT100;
   1:  PR[GP1:91,1] = PR[GP1:90,1] + 4.002;
   1:  PR[GP1:91,2] = PR[GP1:90,2] + -22.370;
   1:L PR[91] R[100]mm/sec CNT100;
   1:  PR[GP1:91,1] = PR[GP1:90,1] + 6.956;
   1:  PR[GP1:91,2] = PR[GP1:90,2] + -25.800;
   1:L PR[91] R[100]mm/sec CNT100;
   1:  PR[GP1:91,1] = PR[GP1:90,1] + 10.914;
   1:  PR[GP1:91,2] = PR[GP1:90,2] + -28.897;
   1:L PR[91] R[100]mm/sec CNT100;
   1:  PR[GP1:91,1] = PR[GP1:90,1] + 11.786;
   1:  PR[GP1:91,2] = PR[GP1:90,2] + -29.531;
   1:L PR[91] R[100]mm/sec CNT100;
   1:  PR[GP1:91,1] = PR[GP1:90,1] + 17.307;
   1:  PR[GP1:91,2] = PR[GP1:90,2] + -32.412;
   1:L PR[91] R[100]mm/sec CNT100;
   1:  PR[GP1:91,1] = PR[GP1:90,1] + 24.197;
   1:  PR[GP1:91,2] = PR[GP1:90,2] + -34.629;
   1:L PR[91] R[100]mm/sec CNT100;
   1:  PR[GP1:91,1] = PR[GP1:90,1] + 25.257;
   1:  PR[GP1:91,2] = PR[GP1:90,2] + -34.768;
   1:L PR[91] R[100]mm/sec CNT100;
   1:  PR[GP1:91,1] = PR[GP1:90,1] + 30.154;
   1:  PR[GP1:91,2] = PR[GP1:90,2] + -35.484;
   1:L PR[91] R[100]mm/sec CNT100;
   1:  PR[GP1:91,1] = PR[GP1:90,1] + 31.958;
   1:  PR[GP1:91,2] = PR[GP1:90,2] + -35.576;
   1:L PR[91] R[100]mm/sec CNT100;
   1:  PR[GP1:91,1] = PR[GP1:90,1] + 37.320;
   1:  PR[GP1:91,2] = PR[GP1:90,2] + -35.427;
   1:L PR[91] R[100]mm/sec CNT100;
   1:  PR[GP1:91,1] = PR[GP1:90,1] + 41.853;
   1:  PR[GP1:91,2] = PR[GP1:90,2] + -34.372;
   1:L PR[91] R[100]mm/sec CNT100;
   1:  PR[GP1:91,1] = PR[GP1:90,1] + 45.993;
   1:  PR[GP1:91,2] = PR[GP1:90,2] + -33.477;
   1:L PR[91] R[100]mm/sec CNT100;
   1:  PR[GP1:91,1] = PR[GP1:90,1] + 48.652;
   1:  PR[GP1:91,2] = PR[GP1:90,2] + -32.436;
   1:L PR[91] R[100]mm/sec CNT100;
   1:  PR[GP1:91,1] = PR[GP1:90,1] + 55.288;
   1:  PR[GP1:91,2] = PR[GP1:90,2] + -28.666;
   1:L PR[91] R[100]mm/sec CNT100;
   1:  PR[GP1:91,1] = PR[GP1:90,1] + 56.797;
   1:  PR[GP1:91,2] = PR[GP1:90,2] + -27.736;
   1:L PR[91] R[100]mm/sec CNT100;
   1:  PR[GP1:91,1] = PR[GP1:90,1] + 57.765;
   1:  PR[GP1:91,2] = PR[GP1:90,2] + -26.871;
   1:L PR[91] R[100]mm/sec CNT100;
   1:  PR[GP1:91,1] = PR[GP1:90,1] + 64.134;
   1:  PR[GP1:91,2] = PR[GP1:90,2] + -20.154;
   1:L PR[91] R[100]mm/sec CNT100;
   1:  PR[GP1:91,1] = PR[GP1:90,1] + 64.431;
   1:  PR[GP1:91,2] = PR[GP1:90,2] + -19.769;
   1:L PR[91] R[100]mm/sec CNT100;
   1:  PR[GP1:91,1] = PR[GP1:90,1] + 69.105;
   1:  PR[GP1:91,2] = PR[GP1:90,2] + -10.461;
   1:L PR[91] R[100]mm/sec CNT100;
   1:  PR[GP1:91,1] = PR[GP1:90,1] + 70.694;
   1:  PR[GP1:91,2] = PR[GP1:90,2] + -0.072;
   1:L PR[91] R[100]mm/sec CNT100;
   1:  PR[GP1:91,1] = PR[GP1:90,1] + 69.105;
   1:  PR[GP1:91,2] = PR[GP1:90,2] + 10.317;
   1:L PR[91] R[100]mm/sec CNT100;
   1:  PR[GP1:91,1] = PR[GP1:90,1] + 64.431;
   1:  PR[GP1:91,2] = PR[GP1:90,2] + 19.625;
   1:L PR[91] R[100]mm/sec CNT100;
   1:  PR[GP1:91,1] = PR[GP1:90,1] + 64.134;
   1:  PR[GP1:91,2] = PR[GP1:90,2] + 20.009;
   1:L PR[91] R[100]mm/sec CNT100;
   1:  PR[GP1:91,1] = PR[GP1:90,1] + 57.765;
   1:  PR[GP1:91,2] = PR[GP1:90,2] + 26.727;
   1:L PR[91] R[100]mm/sec CNT100;
   1:  PR[GP1:91,1] = PR[GP1:90,1] + 56.806;
   1:  PR[GP1:91,2] = PR[GP1:90,2] + 27.583;
   1:L PR[91] R[100]mm/sec CNT100;
   1:  PR[GP1:91,1] = PR[GP1:90,1] + 50.461;
   1:  PR[GP1:91,2] = PR[GP1:90,2] + 31.149;
   1:L PR[91] R[100]mm/sec CNT100;
   1:  PR[GP1:91,1] = PR[GP1:90,1] + 48.639;
   1:  PR[GP1:91,2] = PR[GP1:90,2] + 32.297;
   1:L PR[91] R[100]mm/sec CNT100;
   1:  PR[GP1:91,1] = PR[GP1:90,1] + 45.988;
   1:  PR[GP1:91,2] = PR[GP1:90,2] + 33.335;
   1:L PR[91] R[100]mm/sec CNT100;
   1:  PR[GP1:91,1] = PR[GP1:90,1] + 40.971;
   1:  PR[GP1:91,2] = PR[GP1:90,2] + 34.517;
   1:L PR[91] R[100]mm/sec CNT100;
   1:  PR[GP1:91,1] = PR[GP1:90,1] + 37.327;
   1:  PR[GP1:91,2] = PR[GP1:90,2] + 35.283;
   1:L PR[91] R[100]mm/sec CNT100;
   1:  PR[GP1:91,1] = PR[GP1:90,1] + 31.958;
   1:  PR[GP1:91,2] = PR[GP1:90,2] + 35.432;
   1:L PR[91] R[100]mm/sec CNT100;
   1:  PR[GP1:91,1] = PR[GP1:90,1] + 30.154;
   1:  PR[GP1:91,2] = PR[GP1:90,2] + 35.340;
   1:L PR[91] R[100]mm/sec CNT100;
   1:  PR[GP1:91,1] = PR[GP1:90,1] + 25.257;
   1:  PR[GP1:91,2] = PR[GP1:90,2] + 34.624;
   1:L PR[91] R[100]mm/sec CNT100;
   1:  PR[GP1:91,1] = PR[GP1:90,1] + 24.196;
   1:  PR[GP1:91,2] = PR[GP1:90,2] + 34.484;
   1:L PR[91] R[100]mm/sec CNT100;
   1:  PR[GP1:91,1] = PR[GP1:90,1] + 18.126;
   1:  PR[GP1:91,2] = PR[GP1:90,2] + 32.553;
   1:L PR[91] R[100]mm/sec CNT100;
   1:  PR[GP1:91,1] = PR[GP1:90,1] + 17.314;
   1:  PR[GP1:91,2] = PR[GP1:90,2] + 32.272;
   1:L PR[91] R[100]mm/sec CNT100;
   1:  PR[GP1:91,1] = PR[GP1:90,1] + 11.784;
   1:  PR[GP1:91,2] = PR[GP1:90,2] + 29.386;
   1:L PR[91] R[100]mm/sec CNT100;
   1:  PR[GP1:91,1] = PR[GP1:90,1] + 11.162;
   1:  PR[GP1:91,2] = PR[GP1:90,2] + 28.946;
   1:L PR[91] R[100]mm/sec CNT100;
   1:  PR[GP1:91,1] = PR[GP1:90,1] + 7.093;
   1:  PR[GP1:91,2] = PR[GP1:90,2] + 25.762;
   1:L PR[91] R[100]mm/sec CNT100;
   1:  PR[GP1:91,1] = PR[GP1:90,1] + 3.984;
   1:  PR[GP1:91,2] = PR[GP1:90,2] + 22.144;
   1:L PR[91] R[100]mm/sec CNT100;
   1:  PR[GP1:91,1] = PR[GP1:90,1] + 3.312;
   1:  PR[GP1:91,2] = PR[GP1:90,2] + 21.878;
   1:L PR[91] R[100]mm/sec CNT100;
   1:  PR[GP1:91,1] = PR[GP1:90,1] + 0.547;
   1:  PR[GP1:91,2] = PR[GP1:90,2] + 20.465;
   1:L PR[91] R[100]mm/sec CNT100;
   1:  ! -- Layer/Ebene 71 -- !;
   1:  PR[91] = PR[90];
   1:  PR[GP1:91,1] = PR[GP1:90,1] + -0.857;
   1:  PR[GP1:91,2] = PR[GP1:90,2] + 20.981;
   1:  PR[GP1:91,3] = PR[GP1:90,3] + 43.615;
   1:L PR[91] R[100]mm/sec CNT100;
   1:  PR[GP1:91,1] = PR[GP1:90,1] + -3.752;
   1:  PR[GP1:91,2] = PR[GP1:90,2] + 22.454;
   1:L PR[91] R[100]mm/sec CNT100;
   1:  PR[GP1:91,1] = PR[GP1:90,1] + -6.687;
   1:  PR[GP1:91,2] = PR[GP1:90,2] + 25.866;
   1:L PR[91] R[100]mm/sec CNT100;
   1:  PR[GP1:91,1] = PR[GP1:90,1] + -10.602;
   1:  PR[GP1:91,2] = PR[GP1:90,2] + 28.932;
   1:L PR[91] R[100]mm/sec CNT100;
   1:  PR[GP1:91,1] = PR[GP1:90,1] + -11.342;
   1:  PR[GP1:91,2] = PR[GP1:90,2] + 29.455;
   1:L PR[91] R[100]mm/sec CNT100;
   1:  PR[GP1:91,1] = PR[GP1:90,1] + -16.769;
   1:  PR[GP1:91,2] = PR[GP1:90,2] + 32.294;
   1:L PR[91] R[100]mm/sec CNT100;
   1:  PR[GP1:91,1] = PR[GP1:90,1] + -23.791;
   1:  PR[GP1:91,2] = PR[GP1:90,2] + 34.561;
   1:L PR[91] R[100]mm/sec CNT100;
   1:  PR[GP1:91,1] = PR[GP1:90,1] + -27.280;
   1:  PR[GP1:91,2] = PR[GP1:90,2] + 35.017;
   1:L PR[91] R[100]mm/sec CNT100;
   1:  PR[GP1:91,1] = PR[GP1:90,1] + -30.091;
   1:  PR[GP1:91,2] = PR[GP1:90,2] + 35.426;
   1:L PR[91] R[100]mm/sec CNT100;
   1:  PR[GP1:91,1] = PR[GP1:90,1] + -31.107;
   1:  PR[GP1:91,2] = PR[GP1:90,2] + 35.477;
   1:L PR[91] R[100]mm/sec CNT100;
   1:  PR[GP1:91,1] = PR[GP1:90,1] + -37.015;
   1:  PR[GP1:91,2] = PR[GP1:90,2] + 35.309;
   1:L PR[91] R[100]mm/sec CNT100;
   1:  PR[GP1:91,1] = PR[GP1:90,1] + -40.670;
   1:  PR[GP1:91,2] = PR[GP1:90,2] + 34.460;
   1:L PR[91] R[100]mm/sec CNT100;
   1:  PR[GP1:91,1] = PR[GP1:90,1] + -45.409;
   1:  PR[GP1:91,2] = PR[GP1:90,2] + 33.433;
   1:L PR[91] R[100]mm/sec CNT100;
   1:  PR[GP1:91,1] = PR[GP1:90,1] + -48.455;
   1:  PR[GP1:91,2] = PR[GP1:90,2] + 32.234;
   1:L PR[91] R[100]mm/sec CNT100;
   1:  PR[GP1:91,1] = PR[GP1:90,1] + -54.462;
   1:  PR[GP1:91,2] = PR[GP1:90,2] + 28.816;
   1:L PR[91] R[100]mm/sec CNT100;
   1:  PR[GP1:91,1] = PR[GP1:90,1] + -56.385;
   1:  PR[GP1:91,2] = PR[GP1:90,2] + 27.625;
   1:L PR[91] R[100]mm/sec CNT100;
   1:  PR[GP1:91,1] = PR[GP1:90,1] + -57.623;
   1:  PR[GP1:91,2] = PR[GP1:90,2] + 26.515;
   1:L PR[91] R[100]mm/sec CNT100;
   1:  PR[GP1:91,1] = PR[GP1:90,1] + -63.563;
   1:  PR[GP1:91,2] = PR[GP1:90,2] + 20.270;
   1:L PR[91] R[100]mm/sec CNT100;
   1:  PR[GP1:91,1] = PR[GP1:90,1] + -64.096;
   1:  PR[GP1:91,2] = PR[GP1:90,2] + 19.578;
   1:L PR[91] R[100]mm/sec CNT100;
